KUKA KRL program: f1_Kuka_APT210T02S10.SRC

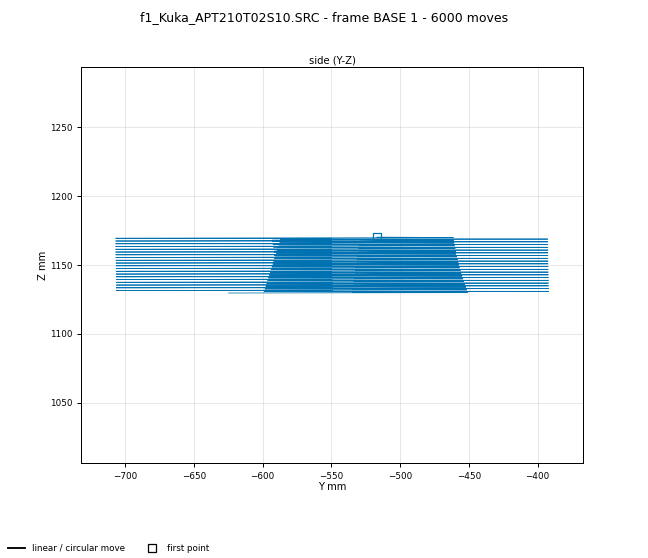
[picture p0: tool path of f1_Kuka_APT210T02S10.SRC in frame BASE 1, 6000 of 6001 moves have a stored position in this frame; points joined in program order, loops and branches not executed]
&ACCESS RVP
&REL 2
&PARAM TEMPLATE = C:\KRC\Roboter\Template\vorgabe
&PARAM EDITMASK = *
DEF f1_Kuka_APT210T02S10()


;FOLD INI;%{PE}%V3.2.0,%MKUKATPBASIS,%CINIT,%VCOMMON,%P
  ;FOLD BAS INI;%{E}%V3.2.0,%MKUKATPBASIS,%CINIT,%VINIT,%P
    GLOBAL INTERRUPT DECL 3 WHEN $STOPMESS==TRUE DO IR_STOPM ( )
    INTERRUPT ON 3
    BAS (#INITMOV,0 )
  ;ENDFOLD (BAS INI)
  ;FOLD USER INI;%{E}%V3.2.0,%MKUKATPUSER,%CINIT,%VINIT,%P
    ;Make your modifications here
  ;ENDFOLD (USER INI)
;ENDFOLD (INI)


;*** Make Null PTP Move
  PTP $pos_act

;*** Auto Load The Correct TOOL Data
  $tool=tool_data[2]

;*** Auto Load The Correct BASE Data
  $base=base_data[1]

  $ADVANCE = 5

;*** Restate Last Velocity
MMPM(30000.0)
SetRPM(8000)
LIN {X -0.168,Y -516.836,Z 1170.287,A 0.000,B 0.000,C 90.000,E1 267.593} C_DIS
LIN {X 0.032,Y -515.961,Z 1170.278,A 0.000,B 0.000,C 90.000,E1 266.102} C_DIS
LIN {X -0.268,Y -514.882,Z 1170.270,A 0.000,B 0.000,C 90.000,E1 264.666} C_DIS
LIN {X -0.155,Y -513.023,Z 1170.259,A 0.000,B 0.000,C 90.000,E1 262.591} C_DIS
LIN {X 0.153,Y -511.888,Z 1170.252,A 0.000,B 0.000,C 90.000,E1 261.376} C_DIS
LIN {X -0.212,Y -509.655,Z 1170.239,A 0.000,B 0.000,C 90.000,E1 259.050} C_DIS
LIN {X 0.192,Y -508.384,Z 1170.231,A 0.000,B 0.000,C 90.000,E1 257.521} C_DIS
LIN {X -0.015,Y -506.651,Z 1170.219,A 0.000,B 0.000,C 90.000,E1 255.463} C_DIS
LIN {X -0.094,Y -505.142,Z 1170.209,A 0.000,B 0.000,C 90.000,E1 253.685} C_DIS
LIN {X 0.005,Y -503.268,Z 1170.198,A 0.000,B 0.000,C 90.000,E1 251.583} C_DIS
LIN {X 0.305,Y -501.633,Z 1170.188,A 0.000,B 0.000,C 90.000,E1 249.752} C_DIS
LIN {X 0.102,Y -499.916,Z 1170.178,A 0.000,B 0.000,C 90.000,E1 247.975} C_DIS
LIN {X -0.084,Y -498.784,Z 1170.171,A 0.000,B 0.000,C 90.000,E1 246.794} C_DIS
LIN {X 0.030,Y -496.635,Z 1170.161,A 0.000,B 0.000,C 90.000,E1 244.973} C_DIS
LIN {X -0.003,Y -495.127,Z 1170.154,A 0.000,B 0.000,C 90.000,E1 243.768} C_DIS
LIN {X -0.213,Y -492.694,Z 1170.144,A 0.000,B 0.000,C 90.000,E1 241.975} C_DIS
LIN {X 0.240,Y -489.792,Z 1170.132,A 0.000,B 0.000,C 90.000,E1 239.793} C_DIS
LIN {X -0.045,Y -487.193,Z 1170.122,A 0.000,B 0.000,C 90.000,E1 237.995} C_DIS
LIN {X 0.307,Y -484.902,Z 1170.114,A 0.000,B 0.000,C 90.000,E1 236.421} C_DIS
LIN {X -0.151,Y -481.804,Z 1170.102,A 0.000,B 0.000,C 90.000,E1 234.322} C_DIS
LIN {X 0.167,Y -480.053,Z 1170.095,A 0.000,B 0.000,C 90.000,E1 233.050} C_DIS
LIN {X -0.126,Y -477.814,Z 1170.086,A 0.000,B 0.000,C 90.000,E1 231.537} C_DIS
LIN {X -0.166,Y -475.649,Z 1170.078,A 0.000,B 0.000,C 90.000,E1 229.989} C_DIS
LIN {X 0.056,Y -473.594,Z 1170.069,A 0.000,B 0.000,C 90.000,E1 228.405} C_DIS
LIN {X -0.073,Y -472.656,Z 1170.066,A 0.000,B 0.000,C 90.000,E1 227.796} C_DIS
LIN {X 0.019,Y -466.553,Z 1170.043,A 0.000,B 0.000,C 90.000,E1 223.704} C_DIS
LIN {X -0.010,Y -463.777,Z 1170.027,A 0.000,B 0.000,C 90.000,E1 220.862} C_DIS
LIN {X 0.041,Y -462.198,Z 1170.009,A 0.000,B 0.000,C 90.000,E1 217.684} C_DIS
LIN {X -0.051,Y -461.506,Z 1169.997,A 0.000,B 0.000,C 90.000,E1 215.471} C_DIS
LIN {X -0.057,Y -461.302,Z 1169.979,A 0.000,B 0.000,C 90.000,E1 212.291} C_DIS
LIN {X -0.265,Y -463.211,Z 1169.960,A 0.000,B 0.000,C 90.000,E1 208.821} C_DIS
LIN {X 0.242,Y -467.166,Z 1169.937,A 0.000,B 0.000,C 90.000,E1 204.643} C_DIS
LIN {X -0.175,Y -473.967,Z 1169.914,A 0.000,B 0.000,C 90.000,E1 200.610} C_DIS
LIN {X 0.182,Y -481.265,Z 1169.897,A 0.000,B 0.000,C 90.000,E1 197.457} C_DIS
LIN {X 0.057,Y -488.321,Z 1169.883,A 0.000,B 0.000,C 90.000,E1 195.009} C_DIS
LIN {X 0.091,Y -494.167,Z 1169.873,A 0.000,B 0.000,C 90.000,E1 193.175} C_DIS
LIN {X 0.040,Y -500.228,Z 1169.863,A 0.000,B 0.000,C 90.000,E1 191.366} C_DIS
LIN {X 0.024,Y -508.467,Z 1169.850,A 0.000,B 0.000,C 90.000,E1 188.973} C_DIS
LIN {X 0.172,Y -513.875,Z 1169.842,A 0.000,B 0.000,C 90.000,E1 187.473} C_DIS
LIN {X -0.083,Y -519.141,Z 1169.833,A 0.000,B 0.000,C 90.000,E1 186.030} C_DIS
LIN {X 0.214,Y -526.425,Z 1169.822,A 0.000,B 0.000,C 90.000,E1 183.955} C_DIS
LIN {X 0.093,Y -531.627,Z 1169.814,A 0.000,B 0.000,C 90.000,E1 182.522} C_DIS
LIN {X 0.067,Y -536.700,Z 1169.806,A 0.000,B 0.000,C 90.000,E1 181.088} C_DIS
LIN {X 0.146,Y -542.917,Z 1169.797,A 0.000,B 0.000,C 90.000,E1 179.370} C_DIS
LIN {X -0.219,Y -548.050,Z 1169.789,A 0.000,B 0.000,C 90.000,E1 177.993} C_DIS
LIN {X 0.003,Y -552.105,Z 1169.782,A 0.000,B 0.000,C 90.000,E1 176.846} C_DIS
LIN {X -0.088,Y -558.170,Z 1169.773,A 0.000,B 0.000,C 90.000,E1 175.179} C_DIS
LIN {X -0.149,Y -563.203,Z 1169.766,A 0.000,B 0.000,C 90.000,E1 173.799} C_DIS
LIN {X 0.032,Y -569.210,Z 1169.756,A 0.000,B 0.000,C 90.000,E1 172.129} C_DIS
LIN {X -0.066,Y -575.096,Z 1169.747,A 0.000,B 0.000,C 90.000,E1 170.500} C_DIS
LIN {X 0.100,Y -579.011,Z 1169.741,A 0.000,B 0.000,C 90.000,E1 169.398} C_DIS
LIN {X 0.330,Y -584.760,Z 1169.732,A 0.000,B 0.000,C 90.000,E1 167.757} C_DIS
LIN {X 0.109,Y -590.326,Z 1169.723,A 0.000,B 0.000,C 90.000,E1 166.172} C_DIS
LIN {X -0.136,Y -594.851,Z 1169.716,A 0.000,B 0.000,C 90.000,E1 164.866} C_DIS
LIN {X -0.020,Y -600.177,Z 1169.707,A 0.000,B 0.000,C 90.000,E1 163.268} C_DIS
LIN {X -0.023,Y -605.216,Z 1169.698,A 0.000,B 0.000,C 90.000,E1 161.692} C_DIS
LIN {X 0.153,Y -609.204,Z 1169.691,A 0.000,B 0.000,C 90.000,E1 160.369} C_DIS
LIN {X 0.024,Y -613.096,Z 1169.684,A 0.000,B 0.000,C 90.000,E1 159.082} C_DIS
LIN {X -0.011,Y -616.070,Z 1169.678,A 0.000,B 0.000,C 90.000,E1 158.050} C_DIS
LIN {X 0.178,Y -621.128,Z 1169.668,A 0.000,B 0.000,C 90.000,E1 156.230} C_DIS
LIN {X -0.085,Y -624.638,Z 1169.661,A 0.000,B 0.000,C 90.000,E1 154.973} C_DIS
LIN {X -0.002,Y -628.684,Z 1169.652,A 0.000,B 0.000,C 90.000,E1 153.435} C_DIS
LIN {X 0.131,Y -631.934,Z 1169.645,A 0.000,B 0.000,C 90.000,E1 152.153} C_DIS
LIN {X -0.248,Y -635.074,Z 1169.638,A 0.000,B 0.000,C 90.000,E1 150.923} C_DIS
LIN {X -0.271,Y -638.014,Z 1169.631,A 0.000,B 0.000,C 90.000,E1 149.665} C_DIS
LIN {X -0.247,Y -640.798,Z 1169.624,A 0.000,B 0.000,C 90.000,E1 148.408} C_DIS
LIN {X 0.154,Y -643.357,Z 1169.617,A 0.000,B 0.000,C 90.000,E1 147.120} C_DIS
LIN {X 0.059,Y -645.689,Z 1169.610,A 0.000,B 0.000,C 90.000,E1 145.881} C_DIS
LIN {X -0.102,Y -648.344,Z 1169.602,A 0.000,B 0.000,C 90.000,E1 144.402} C_DIS
LIN {X -0.180,Y -650.116,Z 1169.597,A 0.000,B 0.000,C 90.000,E1 143.417} C_DIS
LIN {X -0.314,Y -652.223,Z 1169.590,A 0.000,B 0.000,C 90.000,E1 142.190} C_DIS
LIN {X -0.069,Y -655.747,Z 1169.579,A 0.000,B 0.000,C 90.000,E1 140.194} C_DIS
LIN {X 0.299,Y -658.194,Z 1169.572,A 0.000,B 0.000,C 90.000,E1 138.933} C_DIS
LIN {X 0.206,Y -660.787,Z 1169.565,A 0.000,B 0.000,C 90.000,E1 137.715} C_DIS
LIN {X -0.364,Y -664.336,Z 1169.556,A 0.000,B 0.000,C 90.000,E1 136.053} C_DIS
LIN {X -0.380,Y -669.027,Z 1169.544,A 0.000,B 0.000,C 90.000,E1 133.866} C_DIS
LIN {X -0.255,Y -673.610,Z 1169.533,A 0.000,B 0.000,C 90.000,E1 131.919} C_DIS
LIN {X -0.295,Y -680.008,Z 1169.518,A 0.000,B 0.000,C 90.000,E1 129.277} C_DIS
LIN {X 0.098,Y -683.547,Z 1169.510,A 0.000,B 0.000,C 90.000,E1 127.810} C_DIS
LIN {X -0.031,Y -686.544,Z 1169.504,A 0.000,B 0.000,C 90.000,E1 126.629} C_DIS
LIN {X 0.221,Y -690.089,Z 1169.496,A 0.000,B 0.000,C 90.000,E1 125.185} C_DIS
LIN {X 0.129,Y -692.356,Z 1169.490,A 0.000,B 0.000,C 90.000,E1 124.246} C_DIS
LIN {X -0.110,Y -695.074,Z 1169.484,A 0.000,B 0.000,C 90.000,E1 123.086} C_DIS
LIN {X 0.287,Y -697.651,Z 1169.477,A 0.000,B 0.000,C 90.000,E1 121.878} C_DIS
LIN {X 0.130,Y -699.920,Z 1169.471,A 0.000,B 0.000,C 90.000,E1 120.718} C_DIS
LIN {X -0.021,Y -701.642,Z 1169.466,A 0.000,B 0.000,C 90.000,E1 119.795} C_DIS
LIN {X -0.211,Y -704.040,Z 1169.458,A 0.000,B 0.000,C 90.000,E1 118.409} C_DIS
LIN {X -0.022,Y -705.472,Z 1169.453,A 0.000,B 0.000,C 90.000,E1 117.462} C_DIS
LIN {X 0.224,Y -706.154,Z 1169.449,A 0.000,B 0.000,C 90.000,E1 116.744} C_DIS
LIN {X -0.182,Y -706.639,Z 1169.444,A 0.000,B 0.000,C 90.000,E1 115.848} C_DIS
LIN {X -0.241,Y -706.750,Z 1169.440,A 0.000,B 0.000,C 90.000,E1 115.155} C_DIS
LIN {X 0.348,Y -706.508,Z 1169.437,A 0.000,B 0.000,C 90.000,E1 114.643} C_DIS
LIN {X -0.296,Y -706.272,Z 1169.436,A 0.000,B 0.000,C 90.000,E1 114.463} C_DIS
LIN {X 0.287,Y -705.354,Z 1169.433,A 0.000,B 0.000,C 90.000,E1 113.951} C_DIS
LIN {X -0.354,Y -704.477,Z 1169.432,A 0.000,B 0.000,C 90.000,E1 113.770} C_DIS
LIN {X 0.213,Y -702.290,Z 1169.429,A 0.000,B 0.000,C 90.000,E1 113.259} C_DIS
LIN {X 0.075,Y -701.376,Z 1169.429,A 0.000,B 0.000,C 90.000,E1 113.153} C_DIS
LIN {X -0.030,Y -696.702,Z 1169.426,A 0.000,B 0.000,C 90.000,E1 112.695} C_DIS
LIN {X -0.167,Y -694.978,Z 1169.425,A 0.000,B 0.000,C 90.000,E1 112.589} C_DIS
LIN {X 0.211,Y -692.477,Z 1169.425,A 0.000,B 0.000,C 90.000,E1 112.461} C_DIS
LIN {X -0.061,Y -685.884,Z 1169.424,A 0.000,B 0.000,C 90.000,E1 112.280} C_DIS
LIN {X -0.050,Y -684.884,Z 1169.424,A 0.000,B 0.000,C 90.000,E1 112.259} C_DIS
LIN {X 0.023,Y -677.229,Z 1169.423,A 0.000,B 0.000,C 90.000,E1 112.206} C_DIS
LIN {X -0.028,Y -604.897,Z 1169.423,A 0.000,B 0.000,C 90.000,E1 112.206} C_DIS
LIN {X -0.262,Y -599.969,Z 1169.422,A 0.000,B 0.000,C 90.000,E1 111.897} C_DIS
LIN {X 0.216,Y -595.825,Z 1169.420,A 0.000,B 0.000,C 90.000,E1 111.535} C_DIS
LIN {X 0.002,Y -584.117,Z 1169.414,A 0.000,B 0.000,C 90.000,E1 110.556} C_DIS
LIN {X -0.067,Y -577.421,Z 1169.411,A 0.000,B 0.000,C 90.000,E1 109.993} C_DIS
LIN {X -0.058,Y -574.631,Z 1169.410,A 0.000,B 0.000,C 90.000,E1 109.758} C_DIS
LIN {X -0.102,Y -568.886,Z 1169.407,A 0.000,B 0.000,C 90.000,E1 109.322} C_DIS
LIN {X -0.058,Y -561.036,Z 1169.404,A 0.000,B 0.000,C 90.000,E1 108.779} C_DIS
LIN {X -0.036,Y -556.428,Z 1169.403,A 0.000,B 0.000,C 90.000,E1 108.471} C_DIS
LIN {X 0.260,Y -551.811,Z 1169.401,A 0.000,B 0.000,C 90.000,E1 108.055} C_DIS
LIN {X -0.164,Y -550.478,Z 1169.399,A 0.000,B 0.000,C 90.000,E1 107.873} C_DIS
LIN {X -0.206,Y -550.464,Z 1169.399,A 0.000,B 0.000,C 90.000,E1 107.873} C_DIS
LIN {X 0.054,Y -550.010,Z 1169.397,A 0.000,B 0.000,C 90.000,E1 107.457} C_DIS
LIN {X 0.084,Y -550.645,Z 1169.391,A 0.000,B 0.000,C 90.000,E1 106.441} C_DIS
LIN {X 0.127,Y -551.600,Z 1169.385,A 0.000,B 0.000,C 90.000,E1 105.315} C_DIS
LIN {X 0.139,Y -553.320,Z 1169.374,A 0.000,B 0.000,C 90.000,E1 103.355} C_DIS
LIN {X -0.070,Y -555.144,Z 1169.364,A 0.000,B 0.000,C 90.000,E1 101.422} C_DIS
LIN {X 0.213,Y -557.116,Z 1169.353,A 0.000,B 0.000,C 90.000,E1 99.443} C_DIS
LIN {X -0.156,Y -558.706,Z 1169.343,A 0.000,B 0.000,C 90.000,E1 97.814} C_DIS
LIN {X 0.252,Y -559.602,Z 1169.337,A 0.000,B 0.000,C 90.000,E1 96.663} C_DIS
LIN {X -0.219,Y -560.844,Z 1169.328,A 0.000,B 0.000,C 90.000,E1 95.049} C_DIS
LIN {X 0.164,Y -562.571,Z 1169.314,A 0.000,B 0.000,C 90.000,E1 92.522} C_DIS
LIN {X -0.224,Y -564.025,Z 1169.303,A 0.000,B 0.000,C 90.000,E1 90.630} C_DIS
LIN {X 0.211,Y -564.856,Z 1169.297,A 0.000,B 0.000,C 90.000,E1 89.484} C_DIS
LIN {X 0.216,Y -565.746,Z 1169.290,A 0.000,B 0.000,C 90.000,E1 88.108} C_DIS
LIN {X -0.208,Y -566.791,Z 1169.281,A 0.000,B 0.000,C 90.000,E1 86.502} C_DIS
LIN {X 0.142,Y -568.012,Z 1169.270,A 0.000,B 0.000,C 90.000,E1 84.546} C_DIS
LIN {X -0.151,Y -569.120,Z 1169.261,A 0.000,B 0.000,C 90.000,E1 82.932} C_DIS
LIN {X 0.309,Y -569.631,Z 1169.256,A 0.000,B 0.000,C 90.000,E1 82.064} C_DIS
LIN {X -0.072,Y -570.396,Z 1169.249,A 0.000,B 0.000,C 90.000,E1 80.735} C_DIS
LIN {X 0.206,Y -571.081,Z 1169.241,A 0.000,B 0.000,C 90.000,E1 79.342} C_DIS
LIN {X 0.044,Y -571.783,Z 1169.233,A 0.000,B 0.000,C 90.000,E1 77.993} C_DIS
LIN {X -0.105,Y -572.436,Z 1169.226,A 0.000,B 0.000,C 90.000,E1 76.645} C_DIS
LIN {X -0.108,Y -573.167,Z 1169.218,A 0.000,B 0.000,C 90.000,E1 75.283} C_DIS
LIN {X -0.114,Y -574.441,Z 1169.205,A 0.000,B 0.000,C 90.000,E1 72.834} C_DIS
LIN {X -0.286,Y -575.459,Z 1169.196,A 0.000,B 0.000,C 90.000,E1 71.221} C_DIS
LIN {X -0.072,Y -576.669,Z 1169.187,A 0.000,B 0.000,C 90.000,E1 69.571} C_DIS
LIN {X 0.248,Y -578.771,Z 1169.173,A 0.000,B 0.000,C 90.000,E1 67.102} C_DIS
LIN {X -0.033,Y -579.878,Z 1169.167,A 0.000,B 0.000,C 90.000,E1 66.049} C_DIS
LIN {X 0.188,Y -581.373,Z 1169.158,A 0.000,B 0.000,C 90.000,E1 64.409} C_DIS
LIN {X 0.048,Y -583.149,Z 1169.147,A 0.000,B 0.000,C 90.000,E1 62.538} C_DIS
LIN {X 0.074,Y -584.629,Z 1169.139,A 0.000,B 0.000,C 90.000,E1 60.923} C_DIS
LIN {X -0.101,Y -586.035,Z 1169.130,A 0.000,B 0.000,C 90.000,E1 59.331} C_DIS
LIN {X -0.125,Y -587.060,Z 1169.122,A 0.000,B 0.000,C 90.000,E1 57.995} C_DIS
LIN {X 0.049,Y -588.178,Z 1169.113,A 0.000,B 0.000,C 90.000,E1 56.373} C_DIS
LIN {X -0.184,Y -588.691,Z 1169.109,A 0.000,B 0.000,C 90.000,E1 55.595} C_DIS
LIN {X 0.278,Y -589.415,Z 1169.103,A 0.000,B 0.000,C 90.000,E1 54.482} C_DIS
LIN {X 0.060,Y -590.570,Z 1169.093,A 0.000,B 0.000,C 90.000,E1 52.637} C_DIS
LIN {X -0.032,Y -591.823,Z 1169.081,A 0.000,B 0.000,C 90.000,E1 50.517} C_DIS
LIN {X -0.106,Y -592.247,Z 1169.075,A 0.000,B 0.000,C 90.000,E1 49.461} C_DIS
LIN {X 0.029,Y -592.618,Z 1169.067,A 0.000,B 0.000,C 90.000,E1 48.119} C_DIS
LIN {X 0.122,Y -592.831,Z 1169.060,A 0.000,B 0.000,C 90.000,E1 46.782} C_DIS
LIN {X 0.027,Y -592.788,Z 1169.054,A 0.000,B 0.000,C 90.000,E1 45.729} C_DIS
LIN {X -0.295,Y -592.486,Z 1169.047,A 0.000,B 0.000,C 90.000,E1 44.433} C_DIS
LIN {X -0.159,Y -592.177,Z 1169.042,A 0.000,B 0.000,C 90.000,E1 43.623} C_DIS
LIN {X 0.166,Y -591.591,Z 1169.036,A 0.000,B 0.000,C 90.000,E1 42.528} C_DIS
LIN {X 0.088,Y -590.864,Z 1169.031,A 0.000,B 0.000,C 90.000,E1 41.472} C_DIS
LIN {X 0.005,Y -589.930,Z 1169.025,A 0.000,B 0.000,C 90.000,E1 40.415} C_DIS
LIN {X 0.110,Y -588.475,Z 1169.017,A 0.000,B 0.000,C 90.000,E1 39.072} C_DIS
LIN {X -0.213,Y -587.458,Z 1169.013,A 0.000,B 0.000,C 90.000,E1 38.302} C_DIS
LIN {X -0.256,Y -585.940,Z 1169.007,A 0.000,B 0.000,C 90.000,E1 37.237} C_DIS
LIN {X 0.032,Y -584.075,Z 1169.001,A 0.000,B 0.000,C 90.000,E1 36.137} C_DIS
LIN {X 0.056,Y -582.983,Z 1168.998,A 0.000,B 0.000,C 90.000,E1 35.598} C_DIS
LIN {X -0.050,Y -580.579,Z 1168.992,A 0.000,B 0.000,C 90.000,E1 34.532} C_DIS
LIN {X -0.040,Y -579.112,Z 1168.989,A 0.000,B 0.000,C 90.000,E1 33.992} C_DIS
LIN {X 0.107,Y -574.932,Z 1168.981,A 0.000,B 0.000,C 90.000,E1 32.625} C_DIS
LIN {X 0.084,Y -572.991,Z 1168.978,A 0.000,B 0.000,C 90.000,E1 32.084} C_DIS
LIN {X 0.171,Y -569.582,Z 1168.974,A 0.000,B 0.000,C 90.000,E1 31.258} C_DIS
LIN {X -0.167,Y -565.336,Z 1168.969,A 0.000,B 0.000,C 90.000,E1 30.335} C_DIS
LIN {X 0.032,Y -561.090,Z 1168.964,A 0.000,B 0.000,C 90.000,E1 29.489} C_DIS
LIN {X -0.096,Y -558.078,Z 1168.961,A 0.000,B 0.000,C 90.000,E1 28.949} C_DIS
LIN {X -0.086,Y -552.377,Z 1168.955,A 0.000,B 0.000,C 90.000,E1 27.975} C_DIS
LIN {X 0.086,Y -547.919,Z 1168.952,A 0.000,B 0.000,C 90.000,E1 27.257} C_DIS
LIN {X 0.094,Y -544.067,Z 1168.948,A 0.000,B 0.000,C 90.000,E1 26.693} C_DIS
LIN {X -0.169,Y -539.974,Z 1168.945,A 0.000,B 0.000,C 90.000,E1 26.155} C_DIS
LIN {X -0.214,Y -535.555,Z 1168.942,A 0.000,B 0.000,C 90.000,E1 25.591} C_DIS
LIN {X 0.051,Y -529.716,Z 1168.938,A 0.000,B 0.000,C 90.000,E1 24.847} C_DIS
LIN {X 0.113,Y -523.679,Z 1168.934,A 0.000,B 0.000,C 90.000,E1 24.131} C_DIS
LIN {X 0.093,Y -514.571,Z 1168.929,A 0.000,B 0.000,C 90.000,E1 23.131} C_DIS
LIN {X -0.134,Y -509.137,Z 1168.925,A 0.000,B 0.000,C 90.000,E1 22.589} C_DIS
LIN {X 0.231,Y -500.761,Z 1168.921,A 0.000,B 0.000,C 90.000,E1 21.716} C_DIS
LIN {X 0.086,Y -490.782,Z 1168.916,A 0.000,B 0.000,C 90.000,E1 20.791} C_DIS
LIN {X -0.095,Y -480.589,Z 1168.910,A 0.000,B 0.000,C 90.000,E1 19.885} C_DIS
LIN {X 0.010,Y -470.428,Z 1168.905,A 0.000,B 0.000,C 90.000,E1 18.960} C_DIS
LIN {X -0.086,Y -458.727,Z 1168.900,A 0.000,B 0.000,C 90.000,E1 17.928} C_DIS
LIN {X 0.121,Y -447.291,Z 1168.894,A 0.000,B 0.000,C 90.000,E1 16.858} C_DIS
LIN {X -0.016,Y -428.509,Z 1168.883,A 0.000,B 0.000,C 90.000,E1 15.009} C_DIS
LIN {X -0.007,Y -416.177,Z 1168.876,A 0.000,B 0.000,C 90.000,E1 13.647} C_DIS
LIN {X 0.070,Y -407.100,Z 1168.870,A 0.000,B 0.000,C 90.000,E1 12.535} C_DIS
LIN {X 0.182,Y -399.418,Z 1168.864,A 0.000,B 0.000,C 90.000,E1 11.478} C_DIS
LIN {X 0.126,Y -396.306,Z 1168.861,A 0.000,B 0.000,C 90.000,E1 11.007} C_DIS
LIN {X -0.144,Y -393.394,Z 1168.858,A 0.000,B 0.000,C 90.000,E1 10.423} C_DIS
LIN {X 0.166,Y -392.697,Z 1168.856,A 0.000,B 0.000,C 90.000,E1 10.018} C_DIS
LIN {X 0.128,Y -392.689,Z 1168.856,A 0.000,B 0.000,C 90.000,E1 10.018} C_DIS
LIN {X -0.059,Y -393.219,Z 1168.853,A 0.000,B 0.000,C 90.000,E1 9.613} C_DIS
LIN {X -0.141,Y -394.979,Z 1168.849,A 0.000,B 0.000,C 90.000,E1 8.916} C_DIS
LIN {X 0.138,Y -397.945,Z 1168.845,A 0.000,B 0.000,C 90.000,E1 7.992} C_DIS
LIN {X -0.024,Y -402.282,Z 1168.839,A 0.000,B 0.000,C 90.000,E1 7.004} C_DIS
LIN {X -0.019,Y -407.163,Z 1168.835,A 0.000,B 0.000,C 90.000,E1 6.258} C_DIS
LIN {X 0.161,Y -410.505,Z 1168.833,A 0.000,B 0.000,C 90.000,E1 5.910} C_DIS
LIN {X 0.103,Y -415.574,Z 1168.831,A 0.000,B 0.000,C 90.000,E1 5.511} C_DIS
LIN {X -0.051,Y -426.674,Z 1168.826,A 0.000,B 0.000,C 90.000,E1 4.702} C_DIS
LIN {X 0.136,Y -449.122,Z 1168.817,A 0.000,B 0.000,C 90.000,E1 3.037} C_DIS
LIN {X -0.172,Y -465.211,Z 1168.811,A 0.000,B 0.000,C 90.000,E1 1.949} C_DIS
LIN {X -0.008,Y -474.614,Z 1168.807,A 0.000,B 0.000,C 90.000,E1 1.260} C_DIS
LIN {X 0.001,Y -482.394,Z 1168.804,A 0.000,B 0.000,C 90.000,E1 0.688} C_DIS
LIN {X 0.000,Y -491.215,Z 1168.800,A 0.000,B 0.000,C 90.000,E1 360.000} C_DIS
LIN {X 0.020,Y -496.714,Z 1168.797,A 0.000,B 0.000,C 90.000,E1 359.542} C_DIS
LIN {X -0.079,Y -503.698,Z 1168.794,A 0.000,B 0.000,C 90.000,E1 358.912} C_DIS
LIN {X -0.030,Y -510.446,Z 1168.790,A 0.000,B 0.000,C 90.000,E1 358.224} C_DIS
LIN {X -0.184,Y -516.881,Z 1168.786,A 0.000,B 0.000,C 90.000,E1 357.535} C_DIS
LIN {X -0.024,Y -523.035,Z 1168.782,A 0.000,B 0.000,C 90.000,E1 356.788} C_DIS
LIN {X -0.268,Y -528.498,Z 1168.778,A 0.000,B 0.000,C 90.000,E1 356.102} C_DIS
LIN {X -0.038,Y -533.541,Z 1168.774,A 0.000,B 0.000,C 90.000,E1 355.355} C_DIS
LIN {X -0.021,Y -537.235,Z 1168.771,A 0.000,B 0.000,C 90.000,E1 354.780} C_DIS
LIN {X 0.024,Y -540.612,Z 1168.768,A 0.000,B 0.000,C 90.000,E1 354.204} C_DIS
LIN {X -0.170,Y -544.359,Z 1168.764,A 0.000,B 0.000,C 90.000,E1 353.514} C_DIS
LIN {X 0.273,Y -547.796,Z 1168.760,A 0.000,B 0.000,C 90.000,E1 352.761} C_DIS
LIN {X -0.151,Y -550.453,Z 1168.757,A 0.000,B 0.000,C 90.000,E1 352.243} C_DIS
LIN {X 0.096,Y -553.870,Z 1168.752,A 0.000,B 0.000,C 90.000,E1 351.376} C_DIS
LIN {X -0.211,Y -555.963,Z 1168.749,A 0.000,B 0.000,C 90.000,E1 350.849} C_DIS
LIN {X 0.233,Y -559.687,Z 1168.743,A 0.000,B 0.000,C 90.000,E1 349.690} C_DIS
LIN {X 0.279,Y -562.974,Z 1168.737,A 0.000,B 0.000,C 90.000,E1 348.578} C_DIS
LIN {X -0.176,Y -565.979,Z 1168.731,A 0.000,B 0.000,C 90.000,E1 347.521} C_DIS
LIN {X 0.137,Y -569.476,Z 1168.723,A 0.000,B 0.000,C 90.000,E1 346.117} C_DIS
LIN {X 0.088,Y -572.689,Z 1168.715,A 0.000,B 0.000,C 90.000,E1 344.755} C_DIS
LIN {X 0.257,Y -574.483,Z 1168.711,A 0.000,B 0.000,C 90.000,E1 343.921} C_DIS
LIN {X -0.097,Y -577.404,Z 1168.703,A 0.000,B 0.000,C 90.000,E1 342.598} C_DIS
LIN {X 0.119,Y -579.072,Z 1168.699,A 0.000,B 0.000,C 90.000,E1 341.764} C_DIS
LIN {X 0.027,Y -581.631,Z 1168.691,A 0.000,B 0.000,C 90.000,E1 340.423} C_DIS
LIN {X 0.125,Y -583.415,Z 1168.685,A 0.000,B 0.000,C 90.000,E1 339.337} C_DIS
LIN {X -0.095,Y -584.891,Z 1168.679,A 0.000,B 0.000,C 90.000,E1 338.284} C_DIS
LIN {X -0.165,Y -585.825,Z 1168.675,A 0.000,B 0.000,C 90.000,E1 337.486} C_DIS
LIN {X 0.124,Y -586.340,Z 1168.672,A 0.000,B 0.000,C 90.000,E1 336.922} C_DIS
LIN {X 0.299,Y -586.806,Z 1168.667,A 0.000,B 0.000,C 90.000,E1 336.102} C_DIS
LIN {X -0.179,Y -587.004,Z 1168.664,A 0.000,B 0.000,C 90.000,E1 335.613} C_DIS
LIN {X -0.114,Y -586.849,Z 1168.659,A 0.000,B 0.000,C 90.000,E1 334.537} C_DIS
LIN {X 0.063,Y -586.397,Z 1168.654,A 0.000,B 0.000,C 90.000,E1 333.717} C_DIS
LIN {X 0.092,Y -585.896,Z 1168.651,A 0.000,B 0.000,C 90.000,E1 333.179} C_DIS
LIN {X 0.256,Y -584.870,Z 1168.647,A 0.000,B 0.000,C 90.000,E1 332.359} C_DIS
LIN {X 0.036,Y -582.987,Z 1168.641,A 0.000,B 0.000,C 90.000,E1 331.307} C_DIS
LIN {X -0.206,Y -580.282,Z 1168.635,A 0.000,B 0.000,C 90.000,E1 330.255} C_DIS
LIN {X 0.160,Y -577.838,Z 1168.630,A 0.000,B 0.000,C 90.000,E1 329.410} C_DIS
LIN {X -0.004,Y -574.491,Z 1168.626,A 0.000,B 0.000,C 90.000,E1 328.614} C_DIS
LIN {X 0.181,Y -571.023,Z 1168.622,A 0.000,B 0.000,C 90.000,E1 327.916} C_DIS
LIN {X -0.072,Y -565.352,Z 1168.617,A 0.000,B 0.000,C 90.000,E1 326.993} C_DIS
LIN {X -0.067,Y -562.612,Z 1168.614,A 0.000,B 0.000,C 90.000,E1 326.580} C_DIS
LIN {X 0.129,Y -558.615,Z 1168.611,A 0.000,B 0.000,C 90.000,E1 326.008} C_DIS
LIN {X -0.016,Y -554.424,Z 1168.608,A 0.000,B 0.000,C 90.000,E1 325.468} C_DIS
LIN {X -0.065,Y -551.036,Z 1168.606,A 0.000,B 0.000,C 90.000,E1 325.055} C_DIS
LIN {X 0.097,Y -543.692,Z 1168.601,A 0.000,B 0.000,C 90.000,E1 324.196} C_DIS
LIN {X -0.179,Y -531.199,Z 1168.594,A 0.000,B 0.000,C 90.000,E1 322.844} C_DIS
LIN {X 0.071,Y -525.417,Z 1168.590,A 0.000,B 0.000,C 90.000,E1 322.145} C_DIS
LIN {X 0.185,Y -522.185,Z 1168.587,A 0.000,B 0.000,C 90.000,E1 321.698} C_DIS
LIN {X 0.004,Y -519.752,Z 1168.585,A 0.000,B 0.000,C 90.000,E1 321.251} C_DIS
LIN {X 0.220,Y -517.837,Z 1168.582,A 0.000,B 0.000,C 90.000,E1 320.642} C_DIS
LIN {X -0.097,Y -516.894,Z 1168.577,A 0.000,B 0.000,C 90.000,E1 319.908} C_DIS
LIN {X 0.033,Y -516.898,Z 1168.572,A 0.000,B 0.000,C 90.000,E1 319.013} C_DIS
LIN {X -0.207,Y -517.985,Z 1168.561,A 0.000,B 0.000,C 90.000,E1 316.986} C_DIS
LIN {X 0.107,Y -518.780,Z 1168.553,A 0.000,B 0.000,C 90.000,E1 315.486} C_DIS
LIN {X -0.100,Y -519.889,Z 1168.541,A 0.000,B 0.000,C 90.000,E1 313.461} C_DIS
LIN {X 0.122,Y -521.066,Z 1168.530,A 0.000,B 0.000,C 90.000,E1 311.391} C_DIS
LIN {X 0.138,Y -521.966,Z 1168.522,A 0.000,B 0.000,C 90.000,E1 309.930} C_DIS
LIN {X 0.188,Y -523.013,Z 1168.512,A 0.000,B 0.000,C 90.000,E1 308.177} C_DIS
LIN {X -0.054,Y -524.076,Z 1168.503,A 0.000,B 0.000,C 90.000,E1 306.457} C_DIS
LIN {X 0.076,Y -525.342,Z 1168.490,A 0.000,B 0.000,C 90.000,E1 304.119} C_DIS
LIN {X -0.287,Y -526.458,Z 1168.480,A 0.000,B 0.000,C 90.000,E1 302.418} C_DIS
LIN {X -0.177,Y -527.438,Z 1168.470,A 0.000,B 0.000,C 90.000,E1 300.669} C_DIS
LIN {X -0.119,Y -527.893,Z 1168.465,A 0.000,B 0.000,C 90.000,E1 299.795} C_DIS
LIN {X 0.204,Y -528.484,Z 1168.456,A 0.000,B 0.000,C 90.000,E1 298.025} C_DIS
LIN {X -0.122,Y -528.799,Z 1168.448,A 0.000,B 0.000,C 90.000,E1 296.616} C_DIS
LIN {X -0.141,Y -528.955,Z 1168.441,A 0.000,B 0.000,C 90.000,E1 295.463} C_DIS
LIN {X 0.098,Y -529.006,Z 1168.435,A 0.000,B 0.000,C 90.000,E1 294.283} C_DIS
LIN {X -0.074,Y -528.949,Z 1168.424,A 0.000,B 0.000,C 90.000,E1 292.280} C_DIS
LIN {X -0.148,Y -528.670,Z 1168.414,A 0.000,B 0.000,C 90.000,E1 290.556} C_DIS
LIN {X 0.256,Y -528.273,Z 1168.405,A 0.000,B 0.000,C 90.000,E1 288.779} C_DIS
LIN {X 0.122,Y -527.880,Z 1168.398,A 0.000,B 0.000,C 90.000,E1 287.638} C_DIS
LIN {X -0.001,Y -527.371,Z 1168.390,A 0.000,B 0.000,C 90.000,E1 286.205} C_DIS
LIN {X -0.152,Y -526.839,Z 1168.384,A 0.000,B 0.000,C 90.000,E1 285.064} C_DIS
LIN {X 0.055,Y -526.156,Z 1168.377,A 0.000,B 0.000,C 90.000,E1 283.883} C_DIS
LIN {X 0.268,Y -525.334,Z 1168.369,A 0.000,B 0.000,C 90.000,E1 282.411} C_DIS
LIN {X -0.161,Y -524.370,Z 1168.361,A 0.000,B 0.000,C 90.000,E1 281.007} C_DIS
LIN {X -0.187,Y -523.397,Z 1168.353,A 0.000,B 0.000,C 90.000,E1 279.557} C_DIS
LIN {X -0.225,Y -522.458,Z 1168.345,A 0.000,B 0.000,C 90.000,E1 278.106} C_DIS
LIN {X 0.163,Y -521.408,Z 1168.335,A 0.000,B 0.000,C 90.000,E1 276.315} C_DIS
LIN {X -0.052,Y -520.424,Z 1168.326,A 0.000,B 0.000,C 90.000,E1 274.588} C_DIS
LIN {X 0.189,Y -519.608,Z 1168.316,A 0.000,B 0.000,C 90.000,E1 272.808} C_DIS
LIN {X -0.248,Y -518.576,Z 1168.303,A 0.000,B 0.000,C 90.000,E1 270.516} C_DIS
LIN {X -0.022,Y -517.919,Z 1168.295,A 0.000,B 0.000,C 90.000,E1 269.026} C_DIS
LIN {X -0.250,Y -517.425,Z 1168.288,A 0.000,B 0.000,C 90.000,E1 267.879} C_DIS
LIN {X -0.105,Y -516.392,Z 1168.278,A 0.000,B 0.000,C 90.000,E1 266.102} C_DIS
LIN {X 0.085,Y -515.122,Z 1168.269,A 0.000,B 0.000,C 90.000,E1 264.318} C_DIS
LIN {X 0.208,Y -513.182,Z 1168.257,A 0.000,B 0.000,C 90.000,E1 262.243} C_DIS
LIN {X 0.043,Y -512.324,Z 1168.252,A 0.000,B 0.000,C 90.000,E1 261.376} C_DIS
LIN {X 0.154,Y -509.809,Z 1168.237,A 0.000,B 0.000,C 90.000,E1 258.701} C_DIS
LIN {X 0.104,Y -508.764,Z 1168.231,A 0.000,B 0.000,C 90.000,E1 257.521} C_DIS
LIN {X -0.044,Y -507.309,Z 1168.221,A 0.000,B 0.000,C 90.000,E1 255.755} C_DIS
LIN {X -0.102,Y -505.787,Z 1168.211,A 0.000,B 0.000,C 90.000,E1 253.976} C_DIS
LIN {X -0.067,Y -504.713,Z 1168.204,A 0.000,B 0.000,C 90.000,E1 252.779} C_DIS
LIN {X 0.107,Y -503.060,Z 1168.194,A 0.000,B 0.000,C 90.000,E1 250.967} C_DIS
LIN {X 0.158,Y -501.679,Z 1168.186,A 0.000,B 0.000,C 90.000,E1 249.464} C_DIS
LIN {X 0.132,Y -500.018,Z 1168.176,A 0.000,B 0.000,C 90.000,E1 247.667} C_DIS
LIN {X -0.121,Y -499.139,Z 1168.171,A 0.000,B 0.000,C 90.000,E1 246.794} C_DIS
LIN {X 0.001,Y -496.962,Z 1168.161,A 0.000,B 0.000,C 90.000,E1 244.973} C_DIS
LIN {X 0.018,Y -495.018,Z 1168.153,A 0.000,B 0.000,C 90.000,E1 243.461} C_DIS
LIN {X 0.030,Y -492.590,Z 1168.143,A 0.000,B 0.000,C 90.000,E1 241.641} C_DIS
LIN {X 0.231,Y -490.079,Z 1168.132,A 0.000,B 0.000,C 90.000,E1 239.793} C_DIS
LIN {X 0.191,Y -487.011,Z 1168.120,A 0.000,B 0.000,C 90.000,E1 237.661} C_DIS
LIN {X 0.180,Y -483.775,Z 1168.109,A 0.000,B 0.000,C 90.000,E1 235.515} C_DIS
LIN {X -0.122,Y -481.157,Z 1168.098,A 0.000,B 0.000,C 90.000,E1 233.703} C_DIS
LIN {X 0.084,Y -478.441,Z 1168.088,A 0.000,B 0.000,C 90.000,E1 231.823} C_DIS
LIN {X 0.057,Y -476.206,Z 1168.079,A 0.000,B 0.000,C 90.000,E1 230.275} C_DIS
LIN {X 0.074,Y -473.704,Z 1168.069,A 0.000,B 0.000,C 90.000,E1 228.405} C_DIS
LIN {X 0.039,Y -472.211,Z 1168.064,A 0.000,B 0.000,C 90.000,E1 227.472} C_DIS
LIN {X 0.112,Y -466.186,Z 1168.041,A 0.000,B 0.000,C 90.000,E1 223.380} C_DIS
LIN {X -0.139,Y -463.119,Z 1168.022,A 0.000,B 0.000,C 90.000,E1 219.930} C_DIS
LIN {X 0.061,Y -462.042,Z 1168.009,A 0.000,B 0.000,C 90.000,E1 217.684} C_DIS
LIN {X -0.157,Y -461.368,Z 1167.999,A 0.000,B 0.000,C 90.000,E1 215.804} C_DIS
LIN {X 0.075,Y -461.025,Z 1167.978,A 0.000,B 0.000,C 90.000,E1 211.957} C_DIS
LIN {X -0.279,Y -462.693,Z 1167.960,A 0.000,B 0.000,C 90.000,E1 208.821} C_DIS
LIN {X 0.201,Y -466.585,Z 1167.937,A 0.000,B 0.000,C 90.000,E1 204.643} C_DIS
LIN {X -0.170,Y -472.217,Z 1167.918,A 0.000,B 0.000,C 90.000,E1 201.227} C_DIS
LIN {X 0.071,Y -476.133,Z 1167.907,A 0.000,B 0.000,C 90.000,E1 199.322} C_DIS
LIN {X -0.094,Y -483.327,Z 1167.892,A 0.000,B 0.000,C 90.000,E1 196.551} C_DIS
LIN {X -0.040,Y -492.787,Z 1167.875,A 0.000,B 0.000,C 90.000,E1 193.480} C_DIS
LIN {X -0.091,Y -499.858,Z 1167.863,A 0.000,B 0.000,C 90.000,E1 191.366} C_DIS
LIN {X -0.119,Y -508.171,Z 1167.850,A 0.000,B 0.000,C 90.000,E1 188.973} C_DIS
LIN {X 0.022,Y -513.582,Z 1167.842,A 0.000,B 0.000,C 90.000,E1 187.473} C_DIS
LIN {X -0.160,Y -517.857,Z 1167.835,A 0.000,B 0.000,C 90.000,E1 186.315} C_DIS
LIN {X 0.105,Y -524.111,Z 1167.825,A 0.000,B 0.000,C 90.000,E1 184.531} C_DIS
LIN {X -0.028,Y -529.358,Z 1167.817,A 0.000,B 0.000,C 90.000,E1 183.094} C_DIS
LIN {X -0.108,Y -533.505,Z 1167.811,A 0.000,B 0.000,C 90.000,E1 181.949} C_DIS
LIN {X -0.089,Y -539.726,Z 1167.801,A 0.000,B 0.000,C 90.000,E1 180.229} C_DIS
LIN {X 0.021,Y -544.884,Z 1167.793,A 0.000,B 0.000,C 90.000,E1 178.797} C_DIS
LIN {X 0.190,Y -549.066,Z 1167.787,A 0.000,B 0.000,C 90.000,E1 177.650} C_DIS
LIN {X 0.098,Y -556.173,Z 1167.776,A 0.000,B 0.000,C 90.000,E1 175.698} C_DIS
LIN {X 0.003,Y -561.287,Z 1167.768,A 0.000,B 0.000,C 90.000,E1 174.318} C_DIS
LIN {X 0.147,Y -567.335,Z 1167.759,A 0.000,B 0.000,C 90.000,E1 172.648} C_DIS
LIN {X -0.178,Y -572.356,Z 1167.752,A 0.000,B 0.000,C 90.000,E1 171.310} C_DIS
LIN {X -0.298,Y -578.297,Z 1167.743,A 0.000,B 0.000,C 90.000,E1 169.690} C_DIS
LIN {X -0.088,Y -584.159,Z 1167.734,A 0.000,B 0.000,C 90.000,E1 168.049} C_DIS
LIN {X 0.250,Y -589.739,Z 1167.725,A 0.000,B 0.000,C 90.000,E1 166.408} C_DIS
LIN {X -0.004,Y -594.341,Z 1167.717,A 0.000,B 0.000,C 90.000,E1 165.102} C_DIS
LIN {X 0.106,Y -599.716,Z 1167.708,A 0.000,B 0.000,C 90.000,E1 163.504} C_DIS
LIN {X -0.091,Y -604.769,Z 1167.700,A 0.000,B 0.000,C 90.000,E1 161.945} C_DIS
LIN {X 0.272,Y -608.812,Z 1167.692,A 0.000,B 0.000,C 90.000,E1 160.604} C_DIS
LIN {X -0.121,Y -613.460,Z 1167.684,A 0.000,B 0.000,C 90.000,E1 159.082} C_DIS
LIN {X 0.078,Y -616.393,Z 1167.678,A 0.000,B 0.000,C 90.000,E1 158.028} C_DIS
LIN {X 0.064,Y -619.942,Z 1167.671,A 0.000,B 0.000,C 90.000,E1 156.741} C_DIS
LIN {X -0.224,Y -623.510,Z 1167.664,A 0.000,B 0.000,C 90.000,E1 155.485} C_DIS
LIN {X -0.198,Y -626.258,Z 1167.658,A 0.000,B 0.000,C 90.000,E1 154.460} C_DIS
LIN {X -0.105,Y -629.575,Z 1167.651,A 0.000,B 0.000,C 90.000,E1 153.179} C_DIS
LIN {X 0.075,Y -633.388,Z 1167.643,A 0.000,B 0.000,C 90.000,E1 151.641} C_DIS
LIN {X -0.369,Y -635.222,Z 1167.638,A 0.000,B 0.000,C 90.000,E1 150.923} C_DIS
LIN {X 0.115,Y -637.578,Z 1167.633,A 0.000,B 0.000,C 90.000,E1 149.871} C_DIS
LIN {X 0.131,Y -640.355,Z 1167.626,A 0.000,B 0.000,C 90.000,E1 148.614} C_DIS
LIN {X -0.415,Y -642.426,Z 1167.620,A 0.000,B 0.000,C 90.000,E1 147.661} C_DIS
LIN {X -0.042,Y -644.331,Z 1167.615,A 0.000,B 0.000,C 90.000,E1 146.628} C_DIS
LIN {X -0.118,Y -646.646,Z 1167.608,A 0.000,B 0.000,C 90.000,E1 145.388} C_DIS
LIN {X 0.177,Y -649.729,Z 1167.598,A 0.000,B 0.000,C 90.000,E1 143.623} C_DIS
LIN {X 0.041,Y -651.864,Z 1167.591,A 0.000,B 0.000,C 90.000,E1 142.396} C_DIS
LIN {X -0.237,Y -657.233,Z 1167.575,A 0.000,B 0.000,C 90.000,E1 139.461} C_DIS
LIN {X 0.089,Y -660.781,Z 1167.565,A 0.000,B 0.000,C 90.000,E1 137.715} C_DIS
LIN {X 0.459,Y -664.335,Z 1167.556,A 0.000,B 0.000,C 90.000,E1 135.972} C_DIS
LIN {X -0.008,Y -669.544,Z 1167.542,A 0.000,B 0.000,C 90.000,E1 133.581} C_DIS
LIN {X -0.373,Y -673.577,Z 1167.533,A 0.000,B 0.000,C 90.000,E1 131.919} C_DIS
LIN {X -0.012,Y -679.367,Z 1167.519,A 0.000,B 0.000,C 90.000,E1 129.483} C_DIS
LIN {X -0.025,Y -683.535,Z 1167.510,A 0.000,B 0.000,C 90.000,E1 127.810} C_DIS
LIN {X 0.021,Y -687.100,Z 1167.502,A 0.000,B 0.000,C 90.000,E1 126.377} C_DIS
LIN {X 0.128,Y -690.646,Z 1167.494,A 0.000,B 0.000,C 90.000,E1 124.945} C_DIS
LIN {X -0.137,Y -693.430,Z 1167.488,A 0.000,B 0.000,C 90.000,E1 123.785} C_DIS
LIN {X -0.003,Y -695.595,Z 1167.482,A 0.000,B 0.000,C 90.000,E1 122.832} C_DIS
LIN {X 0.161,Y -697.647,Z 1167.477,A 0.000,B 0.000,C 90.000,E1 121.878} C_DIS
LIN {X 0.003,Y -699.916,Z 1167.471,A 0.000,B 0.000,C 90.000,E1 120.718} C_DIS
LIN {X -0.149,Y -701.609,Z 1167.465,A 0.000,B 0.000,C 90.000,E1 119.795} C_DIS
LIN {X 0.280,Y -704.046,Z 1167.458,A 0.000,B 0.000,C 90.000,E1 118.359} C_DIS
LIN {X -0.151,Y -705.483,Z 1167.453,A 0.000,B 0.000,C 90.000,E1 117.462} C_DIS
LIN {X 0.095,Y -706.160,Z 1167.449,A 0.000,B 0.000,C 90.000,E1 116.744} C_DIS
LIN {X -0.311,Y -706.643,Z 1167.443,A 0.000,B 0.000,C 90.000,E1 115.848} C_DIS
LIN {X -0.370,Y -706.748,Z 1167.440,A 0.000,B 0.000,C 90.000,E1 115.155} C_DIS
LIN {X 0.219,Y -706.475,Z 1167.437,A 0.000,B 0.000,C 90.000,E1 114.643} C_DIS
LIN {X -0.423,Y -706.222,Z 1167.436,A 0.000,B 0.000,C 90.000,E1 114.463} C_DIS
LIN {X 0.159,Y -705.332,Z 1167.433,A 0.000,B 0.000,C 90.000,E1 113.951} C_DIS
LIN {X 0.162,Y -704.429,Z 1167.432,A 0.000,B 0.000,C 90.000,E1 113.718} C_DIS
LIN {X 0.085,Y -702.221,Z 1167.429,A 0.000,B 0.000,C 90.000,E1 113.259} C_DIS
LIN {X -0.053,Y -701.275,Z 1167.429,A 0.000,B 0.000,C 90.000,E1 113.153} C_DIS
LIN {X -0.073,Y -696.704,Z 1167.426,A 0.000,B 0.000,C 90.000,E1 112.695} C_DIS
LIN {X -0.204,Y -694.971,Z 1167.425,A 0.000,B 0.000,C 90.000,E1 112.589} C_DIS
LIN {X 0.180,Y -692.460,Z 1167.425,A 0.000,B 0.000,C 90.000,E1 112.461} C_DIS
LIN {X -0.085,Y -685.888,Z 1167.424,A 0.000,B 0.000,C 90.000,E1 112.280} C_DIS
LIN {X -0.074,Y -684.898,Z 1167.424,A 0.000,B 0.000,C 90.000,E1 112.259} C_DIS
LIN {X -0.106,Y -676.366,Z 1167.423,A 0.000,B 0.000,C 90.000,E1 112.206} C_DIS
LIN {X -0.143,Y -604.673,Z 1167.423,A 0.000,B 0.000,C 90.000,E1 112.206} C_DIS
LIN {X -0.252,Y -599.895,Z 1167.422,A 0.000,B 0.000,C 90.000,E1 111.897} C_DIS
LIN {X 0.225,Y -595.751,Z 1167.420,A 0.000,B 0.000,C 90.000,E1 111.535} C_DIS
LIN {X 0.170,Y -581.356,Z 1167.413,A 0.000,B 0.000,C 90.000,E1 110.301} C_DIS
LIN {X 0.205,Y -574.261,Z 1167.410,A 0.000,B 0.000,C 90.000,E1 109.704} C_DIS
LIN {X -0.022,Y -568.337,Z 1167.407,A 0.000,B 0.000,C 90.000,E1 109.268} C_DIS
LIN {X 0.038,Y -560.438,Z 1167.404,A 0.000,B 0.000,C 90.000,E1 108.725} C_DIS
LIN {X 0.048,Y -555.781,Z 1167.402,A 0.000,B 0.000,C 90.000,E1 108.417} C_DIS
LIN {X 0.254,Y -551.736,Z 1167.401,A 0.000,B 0.000,C 90.000,E1 108.055} C_DIS
LIN {X -0.140,Y -550.422,Z 1167.399,A 0.000,B 0.000,C 90.000,E1 107.873} C_DIS
LIN {X -0.183,Y -550.405,Z 1167.399,A 0.000,B 0.000,C 90.000,E1 107.873} C_DIS
LIN {X -0.196,Y -549.970,Z 1167.397,A 0.000,B 0.000,C 90.000,E1 107.511} C_DIS
LIN {X 0.181,Y -550.378,Z 1167.393,A 0.000,B 0.000,C 90.000,E1 106.732} C_DIS
LIN {X 0.214,Y -551.341,Z 1167.387,A 0.000,B 0.000,C 90.000,E1 105.607} C_DIS
LIN {X 0.214,Y -553.000,Z 1167.376,A 0.000,B 0.000,C 90.000,E1 103.647} C_DIS
LIN {X -0.004,Y -554.786,Z 1167.365,A 0.000,B 0.000,C 90.000,E1 101.715} C_DIS
LIN {X 0.232,Y -556.469,Z 1167.356,A 0.000,B 0.000,C 90.000,E1 100.018} C_DIS
LIN {X 0.262,Y -557.825,Z 1167.348,A 0.000,B 0.000,C 90.000,E1 98.624} C_DIS
LIN {X 0.236,Y -559.086,Z 1167.340,A 0.000,B 0.000,C 90.000,E1 97.239} C_DIS
LIN {X -0.113,Y -560.534,Z 1167.330,A 0.000,B 0.000,C 90.000,E1 95.334} C_DIS
LIN {X -0.152,Y -561.473,Z 1167.322,A 0.000,B 0.000,C 90.000,E1 93.955} C_DIS
LIN {X -0.112,Y -562.681,Z 1167.313,A 0.000,B 0.000,C 90.000,E1 92.293} C_DIS
LIN {X 0.068,Y -564.182,Z 1167.302,A 0.000,B 0.000,C 90.000,E1 90.344} C_DIS
LIN {X -0.060,Y -564.943,Z 1167.296,A 0.000,B 0.000,C 90.000,E1 89.255} C_DIS
LIN {X -0.166,Y -565.666,Z 1167.290,A 0.000,B 0.000,C 90.000,E1 88.165} C_DIS
LIN {X 0.084,Y -566.859,Z 1167.279,A 0.000,B 0.000,C 90.000,E1 86.216} C_DIS
LIN {X -0.297,Y -567.881,Z 1167.270,A 0.000,B 0.000,C 90.000,E1 84.609} C_DIS
LIN {X 0.129,Y -569.185,Z 1167.259,A 0.000,B 0.000,C 90.000,E1 82.648} C_DIS
LIN {X -0.083,Y -570.101,Z 1167.250,A 0.000,B 0.000,C 90.000,E1 81.027} C_DIS
LIN {X -0.183,Y -570.937,Z 1167.241,A 0.000,B 0.000,C 90.000,E1 79.398} C_DIS
LIN {X 0.212,Y -571.610,Z 1167.234,A 0.000,B 0.000,C 90.000,E1 77.993} C_DIS
LIN {X 0.254,Y -572.410,Z 1167.224,A 0.000,B 0.000,C 90.000,E1 76.353} C_DIS
LIN {X 0.247,Y -573.108,Z 1167.217,A 0.000,B 0.000,C 90.000,E1 74.991} C_DIS
LIN {X 0.232,Y -574.450,Z 1167.203,A 0.000,B 0.000,C 90.000,E1 72.543} C_DIS
LIN {X 0.242,Y -575.871,Z 1167.191,A 0.000,B 0.000,C 90.000,E1 70.369} C_DIS
LIN {X 0.089,Y -576.920,Z 1167.184,A 0.000,B 0.000,C 90.000,E1 69.028} C_DIS
LIN {X -0.137,Y -578.624,Z 1167.173,A 0.000,B 0.000,C 90.000,E1 67.155} C_DIS
LIN {X -0.028,Y -579.995,Z 1167.166,A 0.000,B 0.000,C 90.000,E1 65.793} C_DIS
LIN {X 0.197,Y -581.459,Z 1167.157,A 0.000,B 0.000,C 90.000,E1 64.152} C_DIS
LIN {X 0.188,Y -583.002,Z 1167.148,A 0.000,B 0.000,C 90.000,E1 62.538} C_DIS
LIN {X 0.212,Y -584.478,Z 1167.139,A 0.000,B 0.000,C 90.000,E1 60.923} C_DIS
LIN {X 0.035,Y -585.867,Z 1167.130,A 0.000,B 0.000,C 90.000,E1 59.331} C_DIS
LIN {X -0.121,Y -587.053,Z 1167.121,A 0.000,B 0.000,C 90.000,E1 57.740} C_DIS
LIN {X -0.252,Y -588.379,Z 1167.110,A 0.000,B 0.000,C 90.000,E1 55.881} C_DIS
LIN {X -0.077,Y -589.220,Z 1167.103,A 0.000,B 0.000,C 90.000,E1 54.529} C_DIS
LIN {X 0.180,Y -590.372,Z 1167.093,A 0.000,B 0.000,C 90.000,E1 52.637} C_DIS
LIN {X 0.082,Y -591.602,Z 1167.081,A 0.000,B 0.000,C 90.000,E1 50.517} C_DIS
LIN {X -0.203,Y -591.946,Z 1167.076,A 0.000,B 0.000,C 90.000,E1 49.747} C_DIS
LIN {X -0.304,Y -592.389,Z 1167.068,A 0.000,B 0.000,C 90.000,E1 48.162} C_DIS
LIN {X -0.206,Y -592.579,Z 1167.060,A 0.000,B 0.000,C 90.000,E1 46.824} C_DIS
LIN {X 0.128,Y -592.539,Z 1167.054,A 0.000,B 0.000,C 90.000,E1 45.729} C_DIS
LIN {X -0.200,Y -592.216,Z 1167.047,A 0.000,B 0.000,C 90.000,E1 44.433} C_DIS
LIN {X -0.065,Y -591.899,Z 1167.042,A 0.000,B 0.000,C 90.000,E1 43.623} C_DIS
LIN {X 0.255,Y -591.338,Z 1167.036,A 0.000,B 0.000,C 90.000,E1 42.528} C_DIS
LIN {X 0.173,Y -590.599,Z 1167.031,A 0.000,B 0.000,C 90.000,E1 41.472} C_DIS
LIN {X -0.162,Y -589.340,Z 1167.023,A 0.000,B 0.000,C 90.000,E1 40.172} C_DIS
LIN {X -0.271,Y -588.136,Z 1167.017,A 0.000,B 0.000,C 90.000,E1 39.116} C_DIS
LIN {X 0.055,Y -586.755,Z 1167.011,A 0.000,B 0.000,C 90.000,E1 38.016} C_DIS
LIN {X 0.002,Y -585.123,Z 1167.005,A 0.000,B 0.000,C 90.000,E1 36.950} C_DIS
LIN {X -0.067,Y -583.196,Z 1166.999,A 0.000,B 0.000,C 90.000,E1 35.884} C_DIS
LIN {X -0.167,Y -580.733,Z 1166.993,A 0.000,B 0.000,C 90.000,E1 34.818} C_DIS
LIN {X -0.156,Y -579.411,Z 1166.990,A 0.000,B 0.000,C 90.000,E1 34.278} C_DIS
LIN {X 0.171,Y -577.837,Z 1166.987,A 0.000,B 0.000,C 90.000,E1 33.706} C_DIS
LIN {X 0.149,Y -574.440,Z 1166.981,A 0.000,B 0.000,C 90.000,E1 32.625} C_DIS
LIN {X 0.122,Y -572.470,Z 1166.978,A 0.000,B 0.000,C 90.000,E1 32.084} C_DIS
LIN {X 0.082,Y -570.269,Z 1166.975,A 0.000,B 0.000,C 90.000,E1 31.544} C_DIS
LIN {X 0.136,Y -566.642,Z 1166.971,A 0.000,B 0.000,C 90.000,E1 30.718} C_DIS
LIN {X -0.236,Y -564.063,Z 1166.968,A 0.000,B 0.000,C 90.000,E1 30.207} C_DIS
LIN {X 0.121,Y -559.032,Z 1166.962,A 0.000,B 0.000,C 90.000,E1 29.205} C_DIS
LIN {X 0.247,Y -554.245,Z 1166.958,A 0.000,B 0.000,C 90.000,E1 28.359} C_DIS
LIN {X -0.051,Y -550.007,Z 1166.954,A 0.000,B 0.000,C 90.000,E1 27.692} C_DIS
LIN {X -0.154,Y -545.425,Z 1166.950,A 0.000,B 0.000,C 90.000,E1 27.001} C_DIS
LIN {X 0.001,Y -540.395,Z 1166.946,A 0.000,B 0.000,C 90.000,E1 26.283} C_DIS
LIN {X -0.043,Y -536.019,Z 1166.943,A 0.000,B 0.000,C 90.000,E1 25.720} C_DIS
LIN {X -0.258,Y -530.220,Z 1166.939,A 0.000,B 0.000,C 90.000,E1 25.027} C_DIS
LIN {X 0.185,Y -524.143,Z 1166.935,A 0.000,B 0.000,C 90.000,E1 24.259} C_DIS
LIN {X 0.232,Y -516.310,Z 1166.930,A 0.000,B 0.000,C 90.000,E1 23.387} C_DIS
LIN {X 0.042,Y -509.583,Z 1166.926,A 0.000,B 0.000,C 90.000,E1 22.695} C_DIS
LIN {X -0.156,Y -502.694,Z 1166.922,A 0.000,B 0.000,C 90.000,E1 22.025} C_DIS
LIN {X 0.130,Y -492.797,Z 1166.917,A 0.000,B 0.000,C 90.000,E1 21.046} C_DIS
LIN {X 0.234,Y -481.388,Z 1166.911,A 0.000,B 0.000,C 90.000,E1 19.993} C_DIS
LIN {X 0.031,Y -469.573,Z 1166.905,A 0.000,B 0.000,C 90.000,E1 18.960} C_DIS
LIN {X 0.215,Y -457.694,Z 1166.900,A 0.000,B 0.000,C 90.000,E1 17.873} C_DIS
LIN {X -0.114,Y -446.185,Z 1166.894,A 0.000,B 0.000,C 90.000,E1 16.858} C_DIS
LIN {X -0.129,Y -428.823,Z 1166.884,A 0.000,B 0.000,C 90.000,E1 15.134} C_DIS
LIN {X -0.051,Y -413.436,Z 1166.875,A 0.000,B 0.000,C 90.000,E1 13.411} C_DIS
LIN {X 0.053,Y -405.559,Z 1166.869,A 0.000,B 0.000,C 90.000,E1 12.411} C_DIS
LIN {X 0.057,Y -398.051,Z 1166.863,A 0.000,B 0.000,C 90.000,E1 11.366} C_DIS
LIN {X 0.017,Y -395.275,Z 1166.861,A 0.000,B 0.000,C 90.000,E1 10.894} C_DIS
LIN {X -0.074,Y -393.186,Z 1166.858,A 0.000,B 0.000,C 90.000,E1 10.423} C_DIS
LIN {X -0.114,Y -392.633,Z 1166.856,A 0.000,B 0.000,C 90.000,E1 10.074} C_DIS
LIN {X -0.129,Y -393.504,Z 1166.853,A 0.000,B 0.000,C 90.000,E1 9.500} C_DIS
LIN {X 0.195,Y -396.000,Z 1166.848,A 0.000,B 0.000,C 90.000,E1 8.568} C_DIS
LIN {X 0.132,Y -398.447,Z 1166.844,A 0.000,B 0.000,C 90.000,E1 7.871} C_DIS
LIN {X 0.067,Y -401.824,Z 1166.839,A 0.000,B 0.000,C 90.000,E1 7.068} C_DIS
LIN {X 0.063,Y -404.276,Z 1166.837,A 0.000,B 0.000,C 90.000,E1 6.663} C_DIS
LIN {X 0.058,Y -406.471,Z 1166.835,A 0.000,B 0.000,C 90.000,E1 6.315} C_DIS
LIN {X 0.038,Y -407.828,Z 1166.834,A 0.000,B 0.000,C 90.000,E1 6.144} C_DIS
LIN {X 0.203,Y -411.093,Z 1166.832,A 0.000,B 0.000,C 90.000,E1 5.796} C_DIS
LIN {X 0.108,Y -426.523,Z 1166.826,A 0.000,B 0.000,C 90.000,E1 4.645} C_DIS
LIN {X -0.096,Y -445.678,Z 1166.818,A 0.000,B 0.000,C 90.000,E1 3.269} C_DIS
LIN {X 0.011,Y -463.532,Z 1166.811,A 0.000,B 0.000,C 90.000,E1 2.007} C_DIS
LIN {X 0.183,Y -473.030,Z 1166.807,A 0.000,B 0.000,C 90.000,E1 1.318} C_DIS
LIN {X 0.198,Y -482.452,Z 1166.804,A 0.000,B 0.000,C 90.000,E1 0.630} C_DIS
LIN {X 0.000,Y -490.917,Z 1166.800,A 0.000,B 0.000,C 90.000,E1 360.000} C_DIS
LIN {X 0.018,Y -496.419,Z 1166.797,A 0.000,B 0.000,C 90.000,E1 359.542} C_DIS
LIN {X 0.063,Y -503.324,Z 1166.794,A 0.000,B 0.000,C 90.000,E1 358.912} C_DIS
LIN {X 0.141,Y -510.140,Z 1166.790,A 0.000,B 0.000,C 90.000,E1 358.224} C_DIS
LIN {X 0.032,Y -516.646,Z 1166.786,A 0.000,B 0.000,C 90.000,E1 357.535} C_DIS
LIN {X 0.212,Y -522.831,Z 1166.782,A 0.000,B 0.000,C 90.000,E1 356.788} C_DIS
LIN {X 0.003,Y -528.354,Z 1166.778,A 0.000,B 0.000,C 90.000,E1 356.102} C_DIS
LIN {X -0.019,Y -532.508,Z 1166.775,A 0.000,B 0.000,C 90.000,E1 355.527} C_DIS
LIN {X 0.252,Y -537.194,Z 1166.771,A 0.000,B 0.000,C 90.000,E1 354.780} C_DIS
LIN {X 0.032,Y -541.376,Z 1166.767,A 0.000,B 0.000,C 90.000,E1 354.090} C_DIS
LIN {X -0.096,Y -545.097,Z 1166.763,A 0.000,B 0.000,C 90.000,E1 353.394} C_DIS
LIN {X 0.031,Y -549.254,Z 1166.759,A 0.000,B 0.000,C 90.000,E1 352.534} C_DIS
LIN {X 0.131,Y -550.591,Z 1166.757,A 0.000,B 0.000,C 90.000,E1 352.243} C_DIS
LIN {X -0.168,Y -554.017,Z 1166.752,A 0.000,B 0.000,C 90.000,E1 351.432} C_DIS
LIN {X 0.076,Y -556.124,Z 1166.749,A 0.000,B 0.000,C 90.000,E1 350.849} C_DIS
LIN {X -0.028,Y -559.898,Z 1166.743,A 0.000,B 0.000,C 90.000,E1 349.746} C_DIS
LIN {X 0.023,Y -563.201,Z 1166.737,A 0.000,B 0.000,C 90.000,E1 348.634} C_DIS
LIN {X 0.124,Y -566.237,Z 1166.731,A 0.000,B 0.000,C 90.000,E1 347.521} C_DIS
LIN {X -0.109,Y -569.763,Z 1166.723,A 0.000,B 0.000,C 90.000,E1 346.172} C_DIS
LIN {X -0.152,Y -573.003,Z 1166.716,A 0.000,B 0.000,C 90.000,E1 344.810} C_DIS
LIN {X 0.022,Y -574.819,Z 1166.711,A 0.000,B 0.000,C 90.000,E1 343.976} C_DIS
LIN {X -0.125,Y -578.340,Z 1166.702,A 0.000,B 0.000,C 90.000,E1 342.362} C_DIS
LIN {X 0.098,Y -579.984,Z 1166.698,A 0.000,B 0.000,C 90.000,E1 341.529} C_DIS
LIN {X -0.183,Y -582.047,Z 1166.692,A 0.000,B 0.000,C 90.000,E1 340.477} C_DIS
LIN {X -0.076,Y -583.849,Z 1166.686,A 0.000,B 0.000,C 90.000,E1 339.390} C_DIS
LIN {X 0.257,Y -585.382,Z 1166.680,A 0.000,B 0.000,C 90.000,E1 338.284} C_DIS
LIN {X 0.068,Y -586.578,Z 1166.674,A 0.000,B 0.000,C 90.000,E1 337.230} C_DIS
LIN {X 0.011,Y -587.201,Z 1166.669,A 0.000,B 0.000,C 90.000,E1 336.433} C_DIS
LIN {X 0.193,Y -587.564,Z 1166.665,A 0.000,B 0.000,C 90.000,E1 335.613} C_DIS
LIN {X 0.264,Y -587.513,Z 1166.659,A 0.000,B 0.000,C 90.000,E1 334.537} C_DIS
LIN {X -0.078,Y -587.124,Z 1166.654,A 0.000,B 0.000,C 90.000,E1 333.768} C_DIS
LIN {X -0.306,Y -586.662,Z 1166.651,A 0.000,B 0.000,C 90.000,E1 333.256} C_DIS
LIN {X 0.135,Y -585.685,Z 1166.647,A 0.000,B 0.000,C 90.000,E1 332.410} C_DIS
LIN {X -0.103,Y -584.812,Z 1166.644,A 0.000,B 0.000,C 90.000,E1 331.897} C_DIS
LIN {X 0.318,Y -583.233,Z 1166.639,A 0.000,B 0.000,C 90.000,E1 331.051} C_DIS
LIN {X 0.212,Y -581.215,Z 1166.635,A 0.000,B 0.000,C 90.000,E1 330.255} C_DIS
LIN {X 0.087,Y -578.769,Z 1166.630,A 0.000,B 0.000,C 90.000,E1 329.459} C_DIS
LIN {X -0.063,Y -575.608,Z 1166.626,A 0.000,B 0.000,C 90.000,E1 328.663} C_DIS
LIN {X -0.167,Y -572.228,Z 1166.622,A 0.000,B 0.000,C 90.000,E1 327.995} C_DIS
LIN {X 0.070,Y -566.850,Z 1166.617,A 0.000,B 0.000,C 90.000,E1 327.041} C_DIS
LIN {X -0.013,Y -563.184,Z 1166.614,A 0.000,B 0.000,C 90.000,E1 326.501} C_DIS
LIN {X -0.125,Y -559.194,Z 1166.611,A 0.000,B 0.000,C 90.000,E1 325.960} C_DIS
LIN {X -0.085,Y -555.318,Z 1166.608,A 0.000,B 0.000,C 90.000,E1 325.435} C_DIS
LIN {X -0.250,Y -550.688,Z 1166.605,A 0.000,B 0.000,C 90.000,E1 324.895} C_DIS
LIN {X -0.133,Y -545.835,Z 1166.602,A 0.000,B 0.000,C 90.000,E1 324.322} C_DIS
LIN {X -0.130,Y -533.619,Z 1166.594,A 0.000,B 0.000,C 90.000,E1 322.970} C_DIS
LIN {X -0.206,Y -527.341,Z 1166.590,A 0.000,B 0.000,C 90.000,E1 322.271} C_DIS
LIN {X -0.206,Y -524.442,Z 1166.588,A 0.000,B 0.000,C 90.000,E1 321.904} C_DIS
LIN {X -0.236,Y -522.369,Z 1166.587,A 0.000,B 0.000,C 90.000,E1 321.618} C_DIS
LIN {X -0.129,Y -520.146,Z 1166.584,A 0.000,B 0.000,C 90.000,E1 321.170} C_DIS
LIN {X -0.104,Y -518.203,Z 1166.581,A 0.000,B 0.000,C 90.000,E1 320.561} C_DIS
LIN {X -0.090,Y -517.276,Z 1166.577,A 0.000,B 0.000,C 90.000,E1 319.828} C_DIS
LIN {X 0.044,Y -517.287,Z 1166.572,A 0.000,B 0.000,C 90.000,E1 318.933} C_DIS
LIN {X -0.185,Y -518.350,Z 1166.561,A 0.000,B 0.000,C 90.000,E1 316.905} C_DIS
LIN {X 0.137,Y -519.121,Z 1166.552,A 0.000,B 0.000,C 90.000,E1 315.405} C_DIS
LIN {X 0.027,Y -520.050,Z 1166.543,A 0.000,B 0.000,C 90.000,E1 313.662} C_DIS
LIN {X 0.224,Y -521.196,Z 1166.531,A 0.000,B 0.000,C 90.000,E1 311.595} C_DIS
LIN {X 0.187,Y -522.249,Z 1166.522,A 0.000,B 0.000,C 90.000,E1 309.850} C_DIS
LIN {X 0.241,Y -523.289,Z 1166.512,A 0.000,B 0.000,C 90.000,E1 308.096} C_DIS
LIN {X 0.003,Y -524.356,Z 1166.502,A 0.000,B 0.000,C 90.000,E1 306.377} C_DIS
LIN {X 0.136,Y -525.654,Z 1166.489,A 0.000,B 0.000,C 90.000,E1 304.040} C_DIS
LIN {X -0.225,Y -526.764,Z 1166.480,A 0.000,B 0.000,C 90.000,E1 302.339} C_DIS
LIN {X -0.114,Y -527.764,Z 1166.470,A 0.000,B 0.000,C 90.000,E1 300.590} C_DIS
LIN {X 0.098,Y -528.310,Z 1166.464,A 0.000,B 0.000,C 90.000,E1 299.411} C_DIS
LIN {X 0.021,Y -528.853,Z 1166.455,A 0.000,B 0.000,C 90.000,E1 297.975} C_DIS
LIN {X 0.006,Y -529.124,Z 1166.449,A 0.000,B 0.000,C 90.000,E1 296.821} C_DIS
LIN {X -0.003,Y -529.310,Z 1166.443,A 0.000,B 0.000,C 90.000,E1 295.668} C_DIS
LIN {X 0.166,Y -529.360,Z 1166.435,A 0.000,B 0.000,C 90.000,E1 294.207} C_DIS
LIN {X -0.007,Y -529.300,Z 1166.423,A 0.000,B 0.000,C 90.000,E1 292.206} C_DIS
LIN {X -0.083,Y -529.058,Z 1166.414,A 0.000,B 0.000,C 90.000,E1 290.482} C_DIS
LIN {X 0.151,Y -528.634,Z 1166.404,A 0.000,B 0.000,C 90.000,E1 288.725} C_DIS
LIN {X 0.011,Y -528.342,Z 1166.399,A 0.000,B 0.000,C 90.000,E1 287.873} C_DIS
LIN {X 0.059,Y -527.699,Z 1166.390,A 0.000,B 0.000,C 90.000,E1 286.134} C_DIS
LIN {X -0.232,Y -527.164,Z 1166.383,A 0.000,B 0.000,C 90.000,E1 285.009} C_DIS
LIN {X 0.026,Y -526.150,Z 1166.374,A 0.000,B 0.000,C 90.000,E1 283.244} C_DIS
LIN {X 0.206,Y -525.661,Z 1166.369,A 0.000,B 0.000,C 90.000,E1 282.355} C_DIS
LIN {X -0.216,Y -524.705,Z 1166.361,A 0.000,B 0.000,C 90.000,E1 280.950} C_DIS
LIN {X -0.233,Y -523.730,Z 1166.353,A 0.000,B 0.000,C 90.000,E1 279.500} C_DIS
LIN {X -0.262,Y -522.790,Z 1166.345,A 0.000,B 0.000,C 90.000,E1 278.049} C_DIS
LIN {X 0.135,Y -521.744,Z 1166.335,A 0.000,B 0.000,C 90.000,E1 276.258} C_DIS
LIN {X -0.147,Y -520.514,Z 1166.322,A 0.000,B 0.000,C 90.000,E1 273.955} C_DIS
LIN {X 0.123,Y -519.864,Z 1166.314,A 0.000,B 0.000,C 90.000,E1 272.465} C_DIS
LIN {X -0.246,Y -518.983,Z 1166.302,A 0.000,B 0.000,C 90.000,E1 270.458} C_DIS
LIN {X -0.070,Y -518.232,Z 1166.293,A 0.000,B 0.000,C 90.000,E1 268.682} C_DIS
LIN {X 0.222,Y -517.652,Z 1166.286,A 0.000,B 0.000,C 90.000,E1 267.478} C_DIS
LIN {X -0.010,Y -517.004,Z 1166.280,A 0.000,B 0.000,C 90.000,E1 266.331} C_DIS
LIN {X -0.214,Y -516.185,Z 1166.273,A 0.000,B 0.000,C 90.000,E1 265.179} C_DIS
LIN {X 0.117,Y -515.514,Z 1166.268,A 0.000,B 0.000,C 90.000,E1 264.261} C_DIS
LIN {X -0.259,Y -513.577,Z 1166.257,A 0.000,B 0.000,C 90.000,E1 262.243} C_DIS
LIN {X 0.087,Y -512.694,Z 1166.252,A 0.000,B 0.000,C 90.000,E1 261.319} C_DIS
LIN {X -0.293,Y -510.195,Z 1166.237,A 0.000,B 0.000,C 90.000,E1 258.701} C_DIS
LIN {X 0.035,Y -508.407,Z 1166.226,A 0.000,B 0.000,C 90.000,E1 256.589} C_DIS
LIN {X -0.005,Y -506.917,Z 1166.216,A 0.000,B 0.000,C 90.000,E1 254.810} C_DIS
LIN {X -0.017,Y -505.622,Z 1166.207,A 0.000,B 0.000,C 90.000,E1 253.323} C_DIS
LIN {X 0.174,Y -503.971,Z 1166.197,A 0.000,B 0.000,C 90.000,E1 251.511} C_DIS
LIN {X -0.144,Y -502.320,Z 1166.188,A 0.000,B 0.000,C 90.000,E1 249.752} C_DIS
LIN {X -0.257,Y -500.349,Z 1166.176,A 0.000,B 0.000,C 90.000,E1 247.667} C_DIS
LIN {X -0.047,Y -499.446,Z 1166.171,A 0.000,B 0.000,C 90.000,E1 246.741} C_DIS
LIN {X 0.074,Y -497.243,Z 1166.161,A 0.000,B 0.000,C 90.000,E1 244.921} C_DIS
LIN {X -0.132,Y -495.289,Z 1166.152,A 0.000,B 0.000,C 90.000,E1 243.435} C_DIS
LIN {X 0.100,Y -492.844,Z 1166.142,A 0.000,B 0.000,C 90.000,E1 241.591} C_DIS
LIN {X -0.125,Y -490.282,Z 1166.132,A 0.000,B 0.000,C 90.000,E1 239.793} C_DIS
LIN {X 0.015,Y -487.663,Z 1166.122,A 0.000,B 0.000,C 90.000,E1 237.946} C_DIS
LIN {X 0.016,Y -484.418,Z 1166.110,A 0.000,B 0.000,C 90.000,E1 235.801} C_DIS
LIN {X 0.216,Y -481.297,Z 1166.098,A 0.000,B 0.000,C 90.000,E1 233.623} C_DIS
LIN {X -0.247,Y -478.544,Z 1166.088,A 0.000,B 0.000,C 90.000,E1 231.823} C_DIS
LIN {X -0.067,Y -476.721,Z 1166.081,A 0.000,B 0.000,C 90.000,E1 230.561} C_DIS
LIN {X -0.032,Y -474.175,Z 1166.071,A 0.000,B 0.000,C 90.000,E1 228.690} C_DIS
LIN {X -0.058,Y -472.768,Z 1166.065,A 0.000,B 0.000,C 90.000,E1 227.757} C_DIS
LIN {X 0.238,Y -467.360,Z 1166.046,A 0.000,B 0.000,C 90.000,E1 224.271} C_DIS
LIN {X 0.078,Y -464.790,Z 1166.034,A 0.000,B 0.000,C 90.000,E1 222.081} C_DIS
LIN {X 0.023,Y -461.888,Z 1166.009,A 0.000,B 0.000,C 90.000,E1 217.649} C_DIS
LIN {X 0.026,Y -460.917,Z 1165.995,A 0.000,B 0.000,C 90.000,E1 215.105} C_DIS
LIN {X 0.107,Y -460.769,Z 1165.976,A 0.000,B 0.000,C 90.000,E1 211.592} C_DIS
LIN {X -0.096,Y -462.403,Z 1165.958,A 0.000,B 0.000,C 90.000,E1 208.437} C_DIS
LIN {X -0.246,Y -466.489,Z 1165.935,A 0.000,B 0.000,C 90.000,E1 204.335} C_DIS
LIN {X -0.011,Y -472.322,Z 1165.916,A 0.000,B 0.000,C 90.000,E1 200.844} C_DIS
LIN {X -0.162,Y -478.741,Z 1165.900,A 0.000,B 0.000,C 90.000,E1 198.055} C_DIS
LIN {X -0.041,Y -488.549,Z 1165.881,A 0.000,B 0.000,C 90.000,E1 194.647} C_DIS
LIN {X 0.088,Y -492.515,Z 1165.875,A 0.000,B 0.000,C 90.000,E1 193.411} C_DIS
LIN {X 0.017,Y -499.618,Z 1165.863,A 0.000,B 0.000,C 90.000,E1 191.299} C_DIS
LIN {X -0.112,Y -508.020,Z 1165.849,A 0.000,B 0.000,C 90.000,E1 188.916} C_DIS
LIN {X 0.094,Y -513.447,Z 1165.841,A 0.000,B 0.000,C 90.000,E1 187.409} C_DIS
LIN {X -0.155,Y -517.729,Z 1165.835,A 0.000,B 0.000,C 90.000,E1 186.258} C_DIS
LIN {X 0.111,Y -524.045,Z 1165.825,A 0.000,B 0.000,C 90.000,E1 184.473} C_DIS
LIN {X -0.051,Y -530.383,Z 1165.815,A 0.000,B 0.000,C 90.000,E1 182.751} C_DIS
LIN {X -0.101,Y -535.590,Z 1165.807,A 0.000,B 0.000,C 90.000,E1 181.318} C_DIS
LIN {X -0.068,Y -540.809,Z 1165.799,A 0.000,B 0.000,C 90.000,E1 179.885} C_DIS
LIN {X 0.154,Y -548.121,Z 1165.788,A 0.000,B 0.000,C 90.000,E1 177.879} C_DIS
LIN {X -0.116,Y -553.253,Z 1165.781,A 0.000,B 0.000,C 90.000,E1 176.502} C_DIS
LIN {X -0.191,Y -559.426,Z 1165.771,A 0.000,B 0.000,C 90.000,E1 174.837} C_DIS
LIN {X -0.175,Y -564.526,Z 1165.764,A 0.000,B 0.000,C 90.000,E1 173.451} C_DIS
LIN {X 0.036,Y -570.636,Z 1165.754,A 0.000,B 0.000,C 90.000,E1 171.781} C_DIS
LIN {X -0.026,Y -576.653,Z 1165.745,A 0.000,B 0.000,C 90.000,E1 170.151} C_DIS
LIN {X -0.188,Y -581.560,Z 1165.738,A 0.000,B 0.000,C 90.000,E1 168.814} C_DIS
LIN {X 0.177,Y -585.459,Z 1165.732,A 0.000,B 0.000,C 90.000,E1 167.701} C_DIS
LIN {X -0.034,Y -591.090,Z 1165.723,A 0.000,B 0.000,C 90.000,E1 166.117} C_DIS
LIN {X -0.270,Y -595.653,Z 1165.716,A 0.000,B 0.000,C 90.000,E1 164.810} C_DIS
LIN {X 0.146,Y -600.116,Z 1165.708,A 0.000,B 0.000,C 90.000,E1 163.449} C_DIS
LIN {X 0.232,Y -604.338,Z 1165.701,A 0.000,B 0.000,C 90.000,E1 162.127} C_DIS
LIN {X 0.086,Y -607.607,Z 1165.695,A 0.000,B 0.000,C 90.000,E1 161.094} C_DIS
LIN {X -0.069,Y -611.535,Z 1165.688,A 0.000,B 0.000,C 90.000,E1 159.806} C_DIS
LIN {X -0.152,Y -615.349,Z 1165.681,A 0.000,B 0.000,C 90.000,E1 158.518} C_DIS
LIN {X -0.195,Y -619.595,Z 1165.672,A 0.000,B 0.000,C 90.000,E1 156.975} C_DIS
LIN {X 0.087,Y -623.151,Z 1165.665,A 0.000,B 0.000,C 90.000,E1 155.665} C_DIS
LIN {X -0.146,Y -626.548,Z 1165.658,A 0.000,B 0.000,C 90.000,E1 154.409} C_DIS
LIN {X -0.055,Y -629.844,Z 1165.651,A 0.000,B 0.000,C 90.000,E1 153.127} C_DIS
LIN {X 0.090,Y -633.023,Z 1165.644,A 0.000,B 0.000,C 90.000,E1 151.847} C_DIS
LIN {X -0.012,Y -635.434,Z 1165.638,A 0.000,B 0.000,C 90.000,E1 150.845} C_DIS
LIN {X -0.392,Y -637.779,Z 1165.632,A 0.000,B 0.000,C 90.000,E1 149.871} C_DIS
LIN {X -0.041,Y -640.538,Z 1165.625,A 0.000,B 0.000,C 90.000,E1 148.584} C_DIS
LIN {X 0.020,Y -643.039,Z 1165.619,A 0.000,B 0.000,C 90.000,E1 147.327} C_DIS
LIN {X 0.336,Y -645.860,Z 1165.610,A 0.000,B 0.000,C 90.000,E1 145.801} C_DIS
LIN {X 0.183,Y -648.487,Z 1165.602,A 0.000,B 0.000,C 90.000,E1 144.322} C_DIS
LIN {X 0.110,Y -650.224,Z 1165.596,A 0.000,B 0.000,C 90.000,E1 143.336} C_DIS
LIN {X -0.018,Y -652.304,Z 1165.590,A 0.000,B 0.000,C 90.000,E1 142.110} C_DIS
LIN {X 0.225,Y -656.804,Z 1165.576,A 0.000,B 0.000,C 90.000,E1 139.622} C_DIS
LIN {X 0.050,Y -660.338,Z 1165.566,A 0.000,B 0.000,C 90.000,E1 137.919} C_DIS
LIN {X -0.040,Y -663.911,Z 1165.557,A 0.000,B 0.000,C 90.000,E1 136.215} C_DIS
LIN {X -0.057,Y -669.601,Z 1165.542,A 0.000,B 0.000,C 90.000,E1 133.542} C_DIS
LIN {X 0.064,Y -673.622,Z 1165.532,A 0.000,B 0.000,C 90.000,E1 131.838} C_DIS
LIN {X 0.403,Y -678.807,Z 1165.521,A 0.000,B 0.000,C 90.000,E1 129.644} C_DIS
LIN {X 0.212,Y -681.779,Z 1165.514,A 0.000,B 0.000,C 90.000,E1 128.463} C_DIS
LIN {X 0.417,Y -683.595,Z 1165.510,A 0.000,B 0.000,C 90.000,E1 127.729} C_DIS
LIN {X -0.091,Y -687.163,Z 1165.502,A 0.000,B 0.000,C 90.000,E1 126.343} C_DIS
LIN {X 0.174,Y -690.706,Z 1165.494,A 0.000,B 0.000,C 90.000,E1 124.898} C_DIS
LIN {X -0.052,Y -694.065,Z 1165.486,A 0.000,B 0.000,C 90.000,E1 123.499} C_DIS
LIN {X -0.260,Y -696.694,Z 1165.480,A 0.000,B 0.000,C 90.000,E1 122.339} C_DIS
LIN {X -0.091,Y -698.629,Z 1165.474,A 0.000,B 0.000,C 90.000,E1 121.386} C_DIS
LIN {X 0.005,Y -700.818,Z 1165.468,A 0.000,B 0.000,C 90.000,E1 120.207} C_DIS
LIN {X 0.091,Y -703.712,Z 1165.459,A 0.000,B 0.000,C 90.000,E1 118.565} C_DIS
LIN {X -0.300,Y -704.857,Z 1165.455,A 0.000,B 0.000,C 90.000,E1 117.897} C_DIS
LIN {X 0.275,Y -705.515,Z 1165.452,A 0.000,B 0.000,C 90.000,E1 117.385} C_DIS
LIN {X 0.200,Y -706.175,Z 1165.448,A 0.000,B 0.000,C 90.000,E1 116.693} C_DIS
LIN {X -0.200,Y -706.654,Z 1165.443,A 0.000,B 0.000,C 90.000,E1 115.796} C_DIS
LIN {X 0.045,Y -706.725,Z 1165.439,A 0.000,B 0.000,C 90.000,E1 115.079} C_DIS
LIN {X -0.306,Y -706.448,Z 1165.437,A 0.000,B 0.000,C 90.000,E1 114.643} C_DIS
LIN {X -0.013,Y -705.684,Z 1165.434,A 0.000,B 0.000,C 90.000,E1 114.155} C_DIS
LIN {X 0.279,Y -705.223,Z 1165.433,A 0.000,B 0.000,C 90.000,E1 113.898} C_DIS
LIN {X 0.065,Y -702.650,Z 1165.430,A 0.000,B 0.000,C 90.000,E1 113.334} C_DIS
LIN {X 0.205,Y -701.917,Z 1165.429,A 0.000,B 0.000,C 90.000,E1 113.206} C_DIS
LIN {X -0.170,Y -697.439,Z 1165.427,A 0.000,B 0.000,C 90.000,E1 112.770} C_DIS
LIN {X -0.034,Y -696.094,Z 1165.426,A 0.000,B 0.000,C 90.000,E1 112.642} C_DIS
LIN {X 0.100,Y -693.912,Z 1165.425,A 0.000,B 0.000,C 90.000,E1 112.514} C_DIS
LIN {X -0.360,Y -686.970,Z 1165.424,A 0.000,B 0.000,C 90.000,E1 112.333} C_DIS
LIN {X -0.105,Y -684.935,Z 1165.424,A 0.000,B 0.000,C 90.000,E1 112.259} C_DIS
LIN {X -0.131,Y -677.165,Z 1165.423,A 0.000,B 0.000,C 90.000,E1 112.206} C_DIS
LIN {X -0.165,Y -604.562,Z 1165.423,A 0.000,B 0.000,C 90.000,E1 112.206} C_DIS
LIN {X 0.204,Y -599.694,Z 1165.422,A 0.000,B 0.000,C 90.000,E1 111.844} C_DIS
LIN {X 0.123,Y -595.565,Z 1165.420,A 0.000,B 0.000,C 90.000,E1 111.535} C_DIS
LIN {X 0.123,Y -579.831,Z 1165.412,A 0.000,B 0.000,C 90.000,E1 110.174} C_DIS
LIN {X 0.057,Y -574.101,Z 1165.410,A 0.000,B 0.000,C 90.000,E1 109.704} C_DIS
LIN {X -0.151,Y -568.194,Z 1165.407,A 0.000,B 0.000,C 90.000,E1 109.268} C_DIS
LIN {X -0.083,Y -560.293,Z 1165.404,A 0.000,B 0.000,C 90.000,E1 108.725} C_DIS
LIN {X -0.071,Y -555.618,Z 1165.402,A 0.000,B 0.000,C 90.000,E1 108.417} C_DIS
LIN {X 0.147,Y -551.599,Z 1165.400,A 0.000,B 0.000,C 90.000,E1 108.055} C_DIS
LIN {X -0.078,Y -550.390,Z 1165.399,A 0.000,B 0.000,C 90.000,E1 107.873} C_DIS
LIN {X -0.120,Y -550.373,Z 1165.399,A 0.000,B 0.000,C 90.000,E1 107.873} C_DIS
LIN {X 0.223,Y -549.955,Z 1165.397,A 0.000,B 0.000,C 90.000,E1 107.457} C_DIS
LIN {X 0.073,Y -550.367,Z 1165.393,A 0.000,B 0.000,C 90.000,E1 106.732} C_DIS
LIN {X 0.107,Y -551.324,Z 1165.387,A 0.000,B 0.000,C 90.000,E1 105.607} C_DIS
LIN {X 0.106,Y -552.960,Z 1165.376,A 0.000,B 0.000,C 90.000,E1 103.647} C_DIS
LIN {X -0.114,Y -554.737,Z 1165.365,A 0.000,B 0.000,C 90.000,E1 101.715} C_DIS
LIN {X -0.010,Y -556.172,Z 1165.357,A 0.000,B 0.000,C 90.000,E1 100.310} C_DIS
LIN {X 0.150,Y -557.767,Z 1165.348,A 0.000,B 0.000,C 90.000,E1 98.624} C_DIS
LIN {X 0.122,Y -559.004,Z 1165.340,A 0.000,B 0.000,C 90.000,E1 97.239} C_DIS
LIN {X -0.229,Y -560.451,Z 1165.330,A 0.000,B 0.000,C 90.000,E1 95.334} C_DIS
LIN {X 0.290,Y -561.410,Z 1165.322,A 0.000,B 0.000,C 90.000,E1 93.898} C_DIS
LIN {X -0.231,Y -562.627,Z 1165.313,A 0.000,B 0.000,C 90.000,E1 92.293} C_DIS
LIN {X -0.159,Y -563.886,Z 1165.303,A 0.000,B 0.000,C 90.000,E1 90.630} C_DIS
LIN {X 0.163,Y -564.532,Z 1165.299,A 0.000,B 0.000,C 90.000,E1 89.771} C_DIS
LIN {X 0.277,Y -565.605,Z 1165.290,A 0.000,B 0.000,C 90.000,E1 88.108} C_DIS
LIN {X -0.041,Y -566.788,Z 1165.279,A 0.000,B 0.000,C 90.000,E1 86.216} C_DIS
LIN {X 0.141,Y -567.776,Z 1165.270,A 0.000,B 0.000,C 90.000,E1 84.552} C_DIS
LIN {X -0.001,Y -569.076,Z 1165.259,A 0.000,B 0.000,C 90.000,E1 82.648} C_DIS
LIN {X -0.215,Y -569.994,Z 1165.250,A 0.000,B 0.000,C 90.000,E1 81.027} C_DIS
LIN {X 0.242,Y -570.806,Z 1165.241,A 0.000,B 0.000,C 90.000,E1 79.342} C_DIS
LIN {X 0.075,Y -571.471,Z 1165.233,A 0.000,B 0.000,C 90.000,E1 77.993} C_DIS
LIN {X -0.252,Y -572.411,Z 1165.223,A 0.000,B 0.000,C 90.000,E1 76.117} C_DIS
LIN {X 0.084,Y -573.201,Z 1165.214,A 0.000,B 0.000,C 90.000,E1 74.448} C_DIS
LIN {X -0.280,Y -574.493,Z 1165.202,A 0.000,B 0.000,C 90.000,E1 72.308} C_DIS
LIN {X 0.093,Y -576.183,Z 1165.188,A 0.000,B 0.000,C 90.000,E1 69.826} C_DIS
LIN {X 0.004,Y -578.017,Z 1165.176,A 0.000,B 0.000,C 90.000,E1 67.667} C_DIS
LIN {X -0.048,Y -579.630,Z 1165.167,A 0.000,B 0.000,C 90.000,E1 66.049} C_DIS
LIN {X 0.168,Y -581.107,Z 1165.158,A 0.000,B 0.000,C 90.000,E1 64.409} C_DIS
LIN {X 0.020,Y -582.881,Z 1165.147,A 0.000,B 0.000,C 90.000,E1 62.538} C_DIS
LIN {X 0.041,Y -584.359,Z 1165.139,A 0.000,B 0.000,C 90.000,E1 60.923} C_DIS
LIN {X -0.139,Y -585.710,Z 1165.130,A 0.000,B 0.000,C 90.000,E1 59.331} C_DIS
LIN {X -0.168,Y -586.724,Z 1165.122,A 0.000,B 0.000,C 90.000,E1 57.995} C_DIS
LIN {X 0.189,Y -588.052,Z 1165.112,A 0.000,B 0.000,C 90.000,E1 56.087} C_DIS
LIN {X 0.218,Y -589.027,Z 1165.103,A 0.000,B 0.000,C 90.000,E1 54.482} C_DIS
LIN {X -0.010,Y -590.195,Z 1165.093,A 0.000,B 0.000,C 90.000,E1 52.637} C_DIS
LIN {X -0.113,Y -591.404,Z 1165.081,A 0.000,B 0.000,C 90.000,E1 50.517} C_DIS
LIN {X -0.193,Y -591.826,Z 1165.075,A 0.000,B 0.000,C 90.000,E1 49.461} C_DIS
LIN {X 0.331,Y -592.166,Z 1165.067,A 0.000,B 0.000,C 90.000,E1 48.081} C_DIS
LIN {X -0.177,Y -592.322,Z 1165.061,A 0.000,B 0.000,C 90.000,E1 47.067} C_DIS
LIN {X 0.152,Y -592.305,Z 1165.056,A 0.000,B 0.000,C 90.000,E1 45.972} C_DIS
LIN {X 0.055,Y -592.114,Z 1165.050,A 0.000,B 0.000,C 90.000,E1 44.919} C_DIS
LIN {X -0.046,Y -591.753,Z 1165.044,A 0.000,B 0.000,C 90.000,E1 43.866} C_DIS
LIN {X 0.035,Y -591.075,Z 1165.036,A 0.000,B 0.000,C 90.000,E1 42.528} C_DIS
LIN {X -0.051,Y -590.301,Z 1165.030,A 0.000,B 0.000,C 90.000,E1 41.472} C_DIS
LIN {X -0.011,Y -588.991,Z 1165.023,A 0.000,B 0.000,C 90.000,E1 40.135} C_DIS
LIN {X -0.308,Y -587.446,Z 1165.016,A 0.000,B 0.000,C 90.000,E1 38.830} C_DIS
LIN {X -0.184,Y -586.385,Z 1165.011,A 0.000,B 0.000,C 90.000,E1 38.016} C_DIS
LIN {X -0.240,Y -584.700,Z 1165.005,A 0.000,B 0.000,C 90.000,E1 36.950} C_DIS
LIN {X -0.153,Y -583.266,Z 1165.001,A 0.000,B 0.000,C 90.000,E1 36.137} C_DIS
LIN {X 0.044,Y -581.563,Z 1164.996,A 0.000,B 0.000,C 90.000,E1 35.311} C_DIS
LIN {X -0.085,Y -578.874,Z 1164.990,A 0.000,B 0.000,C 90.000,E1 34.246} C_DIS
LIN {X -0.087,Y -577.298,Z 1164.987,A 0.000,B 0.000,C 90.000,E1 33.706} C_DIS
LIN {X -0.116,Y -573.834,Z 1164.981,A 0.000,B 0.000,C 90.000,E1 32.625} C_DIS
LIN {X -0.016,Y -570.738,Z 1164.977,A 0.000,B 0.000,C 90.000,E1 31.799} C_DIS
LIN {X -0.069,Y -568.433,Z 1164.974,A 0.000,B 0.000,C 90.000,E1 31.258} C_DIS
LIN {X 0.161,Y -564.681,Z 1164.969,A 0.000,B 0.000,C 90.000,E1 30.413} C_DIS
LIN {X -0.136,Y -560.464,Z 1164.964,A 0.000,B 0.000,C 90.000,E1 29.617} C_DIS
LIN {X -0.267,Y -557.479,Z 1164.961,A 0.000,B 0.000,C 90.000,E1 29.077} C_DIS
LIN {X -0.045,Y -553.459,Z 1164.958,A 0.000,B 0.000,C 90.000,E1 28.359} C_DIS
LIN {X 0.253,Y -550.068,Z 1164.954,A 0.000,B 0.000,C 90.000,E1 27.769} C_DIS
LIN {X -0.214,Y -546.458,Z 1164.951,A 0.000,B 0.000,C 90.000,E1 27.257} C_DIS
LIN {X -0.091,Y -543.567,Z 1164.949,A 0.000,B 0.000,C 90.000,E1 26.821} C_DIS
LIN {X 0.130,Y -539.410,Z 1164.946,A 0.000,B 0.000,C 90.000,E1 26.232} C_DIS
LIN {X -0.059,Y -533.860,Z 1164.942,A 0.000,B 0.000,C 90.000,E1 25.540} C_DIS
LIN {X 0.274,Y -526.808,Z 1164.937,A 0.000,B 0.000,C 90.000,E1 24.643} C_DIS
LIN {X 0.141,Y -521.750,Z 1164.934,A 0.000,B 0.000,C 90.000,E1 24.079} C_DIS
LIN {X 0.122,Y -515.441,Z 1164.930,A 0.000,B 0.000,C 90.000,E1 23.387} C_DIS
LIN {X -0.016,Y -508.743,Z 1164.926,A 0.000,B 0.000,C 90.000,E1 22.695} C_DIS
LIN {X -0.236,Y -501.819,Z 1164.922,A 0.000,B 0.000,C 90.000,E1 22.025} C_DIS
LIN {X 0.180,Y -492.059,Z 1164.917,A 0.000,B 0.000,C 90.000,E1 21.046} C_DIS
LIN {X 0.123,Y -480.375,Z 1164.911,A 0.000,B 0.000,C 90.000,E1 19.993} C_DIS
LIN {X -0.088,Y -467.172,Z 1164.905,A 0.000,B 0.000,C 90.000,E1 18.833} C_DIS
LIN {X -0.119,Y -452.328,Z 1164.897,A 0.000,B 0.000,C 90.000,E1 17.511} C_DIS
LIN {X 0.158,Y -430.693,Z 1164.886,A 0.000,B 0.000,C 90.000,E1 15.371} C_DIS
LIN {X -0.097,Y -415.228,Z 1164.876,A 0.000,B 0.000,C 90.000,E1 13.703} C_DIS
LIN {X -0.015,Y -407.151,Z 1164.871,A 0.000,B 0.000,C 90.000,E1 12.703} C_DIS
LIN {X 0.007,Y -399.458,Z 1164.865,A 0.000,B 0.000,C 90.000,E1 11.658} C_DIS
LIN {X 0.053,Y -395.215,Z 1164.861,A 0.000,B 0.000,C 90.000,E1 10.950} C_DIS
LIN {X -0.128,Y -393.155,Z 1164.858,A 0.000,B 0.000,C 90.000,E1 10.489} C_DIS
LIN {X -0.166,Y -392.591,Z 1164.856,A 0.000,B 0.000,C 90.000,E1 10.141} C_DIS
LIN {X 0.025,Y -393.177,Z 1164.854,A 0.000,B 0.000,C 90.000,E1 9.670} C_DIS
LIN {X -0.018,Y -393.998,Z 1164.852,A 0.000,B 0.000,C 90.000,E1 9.321} C_DIS
LIN {X -0.142,Y -396.606,Z 1164.847,A 0.000,B 0.000,C 90.000,E1 8.454} C_DIS
LIN {X -0.215,Y -398.427,Z 1164.844,A 0.000,B 0.000,C 90.000,E1 7.936} C_DIS
LIN {X -0.121,Y -401.896,Z 1164.839,A 0.000,B 0.000,C 90.000,E1 7.068} C_DIS
LIN {X -0.103,Y -402.825,Z 1164.838,A 0.000,B 0.000,C 90.000,E1 6.891} C_DIS
LIN {X -0.097,Y -406.746,Z 1164.835,A 0.000,B 0.000,C 90.000,E1 6.258} C_DIS
LIN {X 0.042,Y -409.744,Z 1164.833,A 0.000,B 0.000,C 90.000,E1 5.910} C_DIS
LIN {X 0.186,Y -411.237,Z 1164.832,A 0.000,B 0.000,C 90.000,E1 5.739} C_DIS
LIN {X 0.206,Y -424.963,Z 1164.826,A 0.000,B 0.000,C 90.000,E1 4.702} C_DIS
LIN {X -0.081,Y -441.117,Z 1164.820,A 0.000,B 0.000,C 90.000,E1 3.555} C_DIS
LIN {X 0.069,Y -463.753,Z 1164.811,A 0.000,B 0.000,C 90.000,E1 1.949} C_DIS
LIN {X -0.217,Y -473.229,Z 1164.807,A 0.000,B 0.000,C 90.000,E1 1.318} C_DIS
LIN {X -0.209,Y -482.675,Z 1164.803,A 0.000,B 0.000,C 90.000,E1 0.630} C_DIS
LIN {X 0.000,Y -490.599,Z 1164.800,A 0.000,B 0.000,C 90.000,E1 360.000} C_DIS
LIN {X -0.061,Y -497.523,Z 1164.797,A 0.000,B 0.000,C 90.000,E1 359.427} C_DIS
LIN {X -0.056,Y -503.248,Z 1164.794,A 0.000,B 0.000,C 90.000,E1 358.912} C_DIS
LIN {X 0.026,Y -510.129,Z 1164.790,A 0.000,B 0.000,C 90.000,E1 358.224} C_DIS
LIN {X 0.034,Y -516.573,Z 1164.786,A 0.000,B 0.000,C 90.000,E1 357.535} C_DIS
LIN {X -0.247,Y -522.768,Z 1164.782,A 0.000,B 0.000,C 90.000,E1 356.846} C_DIS
LIN {X -0.100,Y -528.504,Z 1164.778,A 0.000,B 0.000,C 90.000,E1 356.102} C_DIS
LIN {X -0.122,Y -532.678,Z 1164.775,A 0.000,B 0.000,C 90.000,E1 355.527} C_DIS
LIN {X 0.151,Y -537.369,Z 1164.771,A 0.000,B 0.000,C 90.000,E1 354.780} C_DIS
LIN {X -0.069,Y -541.602,Z 1164.767,A 0.000,B 0.000,C 90.000,E1 354.090} C_DIS
LIN {X -0.196,Y -545.364,Z 1164.763,A 0.000,B 0.000,C 90.000,E1 353.394} C_DIS
LIN {X -0.091,Y -548.163,Z 1164.760,A 0.000,B 0.000,C 90.000,E1 352.818} C_DIS
LIN {X -0.225,Y -551.456,Z 1164.756,A 0.000,B 0.000,C 90.000,E1 352.129} C_DIS
LIN {X -0.260,Y -554.316,Z 1164.752,A 0.000,B 0.000,C 90.000,E1 351.432} C_DIS
LIN {X -0.015,Y -556.416,Z 1164.749,A 0.000,B 0.000,C 90.000,E1 350.849} C_DIS
LIN {X -0.114,Y -560.217,Z 1164.743,A 0.000,B 0.000,C 90.000,E1 349.746} C_DIS
LIN {X -0.060,Y -563.551,Z 1164.737,A 0.000,B 0.000,C 90.000,E1 348.634} C_DIS
LIN {X 0.218,Y -567.336,Z 1164.729,A 0.000,B 0.000,C 90.000,E1 347.229} C_DIS
LIN {X 0.000,Y -570.783,Z 1164.722,A 0.000,B 0.000,C 90.000,E1 345.880} C_DIS
LIN {X -0.218,Y -573.401,Z 1164.716,A 0.000,B 0.000,C 90.000,E1 344.810} C_DIS
LIN {X 0.154,Y -575.820,Z 1164.709,A 0.000,B 0.000,C 90.000,E1 343.685} C_DIS
LIN {X 0.199,Y -579.362,Z 1164.700,A 0.000,B 0.000,C 90.000,E1 342.054} C_DIS
LIN {X -0.116,Y -580.977,Z 1164.696,A 0.000,B 0.000,C 90.000,E1 341.275} C_DIS
LIN {X -0.023,Y -583.006,Z 1164.690,A 0.000,B 0.000,C 90.000,E1 340.188} C_DIS
LIN {X -0.051,Y -585.148,Z 1164.682,A 0.000,B 0.000,C 90.000,E1 338.847} C_DIS
LIN {X 0.228,Y -585.924,Z 1164.680,A 0.000,B 0.000,C 90.000,E1 338.284} C_DIS
LIN {X -0.075,Y -587.374,Z 1164.672,A 0.000,B 0.000,C 90.000,E1 336.975} C_DIS
LIN {X -0.124,Y -587.906,Z 1164.668,A 0.000,B 0.000,C 90.000,E1 336.177} C_DIS
LIN {X 0.067,Y -588.168,Z 1164.663,A 0.000,B 0.000,C 90.000,E1 335.357} C_DIS
LIN {X 0.262,Y -588.134,Z 1164.659,A 0.000,B 0.000,C 90.000,E1 334.537} C_DIS
LIN {X -0.075,Y -587.825,Z 1164.654,A 0.000,B 0.000,C 90.000,E1 333.768} C_DIS
LIN {X 0.111,Y -587.072,Z 1164.650,A 0.000,B 0.000,C 90.000,E1 332.948} C_DIS
LIN {X 0.035,Y -586.061,Z 1164.645,A 0.000,B 0.000,C 90.000,E1 332.153} C_DIS
LIN {X 0.347,Y -583.995,Z 1164.639,A 0.000,B 0.000,C 90.000,E1 331.051} C_DIS
LIN {X 0.248,Y -582.015,Z 1164.635,A 0.000,B 0.000,C 90.000,E1 330.255} C_DIS
LIN {X -0.022,Y -580.423,Z 1164.632,A 0.000,B 0.000,C 90.000,E1 329.744} C_DIS
LIN {X -0.011,Y -578.611,Z 1164.629,A 0.000,B 0.000,C 90.000,E1 329.203} C_DIS
LIN {X -0.010,Y -576.521,Z 1164.626,A 0.000,B 0.000,C 90.000,E1 328.663} C_DIS
LIN {X 0.058,Y -574.602,Z 1164.624,A 0.000,B 0.000,C 90.000,E1 328.250} C_DIS
LIN {X 0.031,Y -571.732,Z 1164.621,A 0.000,B 0.000,C 90.000,E1 327.709} C_DIS
LIN {X -0.018,Y -568.686,Z 1164.618,A 0.000,B 0.000,C 90.000,E1 327.168} C_DIS
LIN {X -0.187,Y -564.151,Z 1164.614,A 0.000,B 0.000,C 90.000,E1 326.501} C_DIS
LIN {X -0.087,Y -559.232,Z 1164.610,A 0.000,B 0.000,C 90.000,E1 325.801} C_DIS
LIN {X -0.109,Y -556.128,Z 1164.608,A 0.000,B 0.000,C 90.000,E1 325.388} C_DIS
LIN {X -0.207,Y -549.099,Z 1164.603,A 0.000,B 0.000,C 90.000,E1 324.562} C_DIS
LIN {X 0.083,Y -542.931,Z 1164.599,A 0.000,B 0.000,C 90.000,E1 323.829} C_DIS
LIN {X -0.184,Y -532.896,Z 1164.593,A 0.000,B 0.000,C 90.000,E1 322.763} C_DIS
LIN {X 0.050,Y -526.640,Z 1164.589,A 0.000,B 0.000,C 90.000,E1 322.029} C_DIS
LIN {X 0.046,Y -523.864,Z 1164.587,A 0.000,B 0.000,C 90.000,E1 321.662} C_DIS
LIN {X 0.114,Y -521.120,Z 1164.584,A 0.000,B 0.000,C 90.000,E1 321.170} C_DIS
LIN {X -0.154,Y -519.883,Z 1164.583,A 0.000,B 0.000,C 90.000,E1 320.884} C_DIS
LIN {X 0.122,Y -518.856,Z 1164.581,A 0.000,B 0.000,C 90.000,E1 320.561} C_DIS
LIN {X 0.142,Y -517.720,Z 1164.577,A 0.000,B 0.000,C 90.000,E1 319.828} C_DIS
LIN {X 0.163,Y -517.775,Z 1164.570,A 0.000,B 0.000,C 90.000,E1 318.609} C_DIS
LIN {X 0.049,Y -518.677,Z 1164.560,A 0.000,B 0.000,C 90.000,E1 316.863} C_DIS
LIN {X -0.002,Y -519.407,Z 1164.552,A 0.000,B 0.000,C 90.000,E1 315.405} C_DIS
LIN {X 0.253,Y -520.327,Z 1164.543,A 0.000,B 0.000,C 90.000,E1 313.623} C_DIS
LIN {X 0.098,Y -521.448,Z 1164.531,A 0.000,B 0.000,C 90.000,E1 311.595} C_DIS
LIN {X -0.221,Y -522.319,Z 1164.523,A 0.000,B 0.000,C 90.000,E1 310.172} C_DIS
LIN {X 0.125,Y -523.511,Z 1164.512,A 0.000,B 0.000,C 90.000,E1 308.096} C_DIS
LIN {X -0.109,Y -524.590,Z 1164.502,A 0.000,B 0.000,C 90.000,E1 306.377} C_DIS
LIN {X 0.067,Y -525.714,Z 1164.491,A 0.000,B 0.000,C 90.000,E1 304.326} C_DIS
LIN {X 0.120,Y -527.003,Z 1164.479,A 0.000,B 0.000,C 90.000,E1 302.291} C_DIS
LIN {X -0.209,Y -528.033,Z 1164.470,A 0.000,B 0.000,C 90.000,E1 300.590} C_DIS
LIN {X 0.312,Y -528.517,Z 1164.465,A 0.000,B 0.000,C 90.000,E1 299.667} C_DIS
LIN {X -0.065,Y -529.204,Z 1164.455,A 0.000,B 0.000,C 90.000,E1 297.975} C_DIS
LIN {X -0.248,Y -529.439,Z 1164.451,A 0.000,B 0.000,C 90.000,E1 297.129} C_DIS
LIN {X -0.078,Y -529.682,Z 1164.443,A 0.000,B 0.000,C 90.000,E1 295.668} C_DIS
LIN {X 0.098,Y -529.719,Z 1164.435,A 0.000,B 0.000,C 90.000,E1 294.207} C_DIS
LIN {X -0.066,Y -529.658,Z 1164.423,A 0.000,B 0.000,C 90.000,E1 292.206} C_DIS
LIN {X 0.177,Y -529.521,Z 1164.415,A 0.000,B 0.000,C 90.000,E1 290.737} C_DIS
LIN {X 0.108,Y -529.003,Z 1164.404,A 0.000,B 0.000,C 90.000,E1 288.725} C_DIS
LIN {X -0.013,Y -528.578,Z 1164.398,A 0.000,B 0.000,C 90.000,E1 287.583} C_DIS
LIN {X 0.028,Y -528.029,Z 1164.390,A 0.000,B 0.000,C 90.000,E1 286.134} C_DIS
LIN {X 0.253,Y -527.515,Z 1164.383,A 0.000,B 0.000,C 90.000,E1 284.954} C_DIS
LIN {X 0.009,Y -526.531,Z 1164.374,A 0.000,B 0.000,C 90.000,E1 283.244} C_DIS
LIN {X 0.213,Y -525.820,Z 1164.367,A 0.000,B 0.000,C 90.000,E1 282.063} C_DIS
LIN {X -0.224,Y -525.082,Z 1164.361,A 0.000,B 0.000,C 90.000,E1 280.950} C_DIS
LIN {X -0.233,Y -524.097,Z 1164.353,A 0.000,B 0.000,C 90.000,E1 279.500} C_DIS
LIN {X -0.250,Y -522.987,Z 1164.343,A 0.000,B 0.000,C 90.000,E1 277.757} C_DIS
LIN {X 0.146,Y -521.940,Z 1164.333,A 0.000,B 0.000,C 90.000,E1 275.967} C_DIS
LIN {X -0.121,Y -520.923,Z 1164.322,A 0.000,B 0.000,C 90.000,E1 273.955} C_DIS
LIN {X 0.157,Y -520.283,Z 1164.314,A 0.000,B 0.000,C 90.000,E1 272.465} C_DIS
LIN {X -0.094,Y -519.671,Z 1164.306,A 0.000,B 0.000,C 90.000,E1 271.031} C_DIS
LIN {X 0.099,Y -518.929,Z 1164.296,A 0.000,B 0.000,C 90.000,E1 269.255} C_DIS
LIN {X -0.176,Y -518.286,Z 1164.288,A 0.000,B 0.000,C 90.000,E1 267.822} C_DIS
LIN {X 0.057,Y -517.457,Z 1164.280,A 0.000,B 0.000,C 90.000,E1 266.331} C_DIS
LIN {X -0.140,Y -516.657,Z 1164.273,A 0.000,B 0.000,C 90.000,E1 265.179} C_DIS
LIN {X 0.197,Y -515.975,Z 1164.268,A 0.000,B 0.000,C 90.000,E1 264.261} C_DIS
LIN {X 0.063,Y -515.152,Z 1164.263,A 0.000,B 0.000,C 90.000,E1 263.394} C_DIS
LIN {X -0.221,Y -513.480,Z 1164.254,A 0.000,B 0.000,C 90.000,E1 261.659} C_DIS
LIN {X -0.149,Y -510.897,Z 1164.239,A 0.000,B 0.000,C 90.000,E1 258.993} C_DIS
LIN {X 0.278,Y -509.547,Z 1164.231,A 0.000,B 0.000,C 90.000,E1 257.465} C_DIS
LIN {X 0.189,Y -508.349,Z 1164.222,A 0.000,B 0.000,C 90.000,E1 255.992} C_DIS
LIN {X 0.073,Y -507.089,Z 1164.214,A 0.000,B 0.000,C 90.000,E1 254.519} C_DIS
LIN {X 0.121,Y -506.027,Z 1164.208,A 0.000,B 0.000,C 90.000,E1 253.323} C_DIS
LIN {X 0.154,Y -504.894,Z 1164.201,A 0.000,B 0.000,C 90.000,E1 252.127} C_DIS
LIN {X -0.233,Y -503.581,Z 1164.193,A 0.000,B 0.000,C 90.000,E1 250.678} C_DIS
LIN {X -0.006,Y -502.128,Z 1164.184,A 0.000,B 0.000,C 90.000,E1 249.156} C_DIS
LIN {X -0.092,Y -500.735,Z 1164.176,A 0.000,B 0.000,C 90.000,E1 247.667} C_DIS
LIN {X 0.122,Y -499.810,Z 1164.171,A 0.000,B 0.000,C 90.000,E1 246.741} C_DIS
LIN {X -0.143,Y -497.226,Z 1164.159,A 0.000,B 0.000,C 90.000,E1 244.665} C_DIS
LIN {X 0.095,Y -495.226,Z 1164.151,A 0.000,B 0.000,C 90.000,E1 243.127} C_DIS
LIN {X -0.143,Y -493.191,Z 1164.142,A 0.000,B 0.000,C 90.000,E1 241.641} C_DIS
LIN {X 0.077,Y -490.136,Z 1164.131,A 0.000,B 0.000,C 90.000,E1 239.488} C_DIS
LIN {X 0.045,Y -487.461,Z 1164.120,A 0.000,B 0.000,C 90.000,E1 237.661} C_DIS
LIN {X 0.224,Y -484.696,Z 1164.110,A 0.000,B 0.000,C 90.000,E1 235.801} C_DIS
LIN {X -0.243,Y -481.558,Z 1164.098,A 0.000,B 0.000,C 90.000,E1 233.703} C_DIS
LIN {X 0.062,Y -479.655,Z 1164.091,A 0.000,B 0.000,C 90.000,E1 232.431} C_DIS
LIN {X -0.150,Y -476.902,Z 1164.081,A 0.000,B 0.000,C 90.000,E1 230.598} C_DIS
LIN {X 0.093,Y -474.725,Z 1164.072,A 0.000,B 0.000,C 90.000,E1 229.013} C_DIS
LIN {X -0.152,Y -472.855,Z 1164.065,A 0.000,B 0.000,C 90.000,E1 227.796} C_DIS
LIN {X -0.023,Y -468.306,Z 1164.050,A 0.000,B 0.000,C 90.000,E1 224.960} C_DIS
LIN {X -0.041,Y -464.815,Z 1164.034,A 0.000,B 0.000,C 90.000,E1 222.123} C_DIS
LIN {X -0.150,Y -461.914,Z 1164.011,A 0.000,B 0.000,C 90.000,E1 218.016} C_DIS
LIN {X -0.135,Y -460.671,Z 1163.995,A 0.000,B 0.000,C 90.000,E1 215.152} C_DIS
LIN {X 0.069,Y -460.371,Z 1163.976,A 0.000,B 0.000,C 90.000,E1 211.623} C_DIS
LIN {X -0.150,Y -462.535,Z 1163.953,A 0.000,B 0.000,C 90.000,E1 207.513} C_DIS
LIN {X -0.020,Y -465.441,Z 1163.937,A 0.000,B 0.000,C 90.000,E1 204.643} C_DIS
LIN {X -0.002,Y -471.068,Z 1163.918,A 0.000,B 0.000,C 90.000,E1 201.173} C_DIS
LIN {X -0.046,Y -478.152,Z 1163.900,A 0.000,B 0.000,C 90.000,E1 198.055} C_DIS
LIN {X -0.129,Y -484.212,Z 1163.888,A 0.000,B 0.000,C 90.000,E1 195.898} C_DIS
LIN {X 0.171,Y -491.060,Z 1163.876,A 0.000,B 0.000,C 90.000,E1 193.716} C_DIS
LIN {X 0.093,Y -499.179,Z 1163.863,A 0.000,B 0.000,C 90.000,E1 191.299} C_DIS
LIN {X -0.047,Y -507.614,Z 1163.850,A 0.000,B 0.000,C 90.000,E1 188.916} C_DIS
LIN {X 0.050,Y -514.165,Z 1163.840,A 0.000,B 0.000,C 90.000,E1 187.125} C_DIS
LIN {X -0.204,Y -519.482,Z 1163.832,A 0.000,B 0.000,C 90.000,E1 185.682} C_DIS
LIN {X 0.106,Y -524.791,Z 1163.823,A 0.000,B 0.000,C 90.000,E1 184.188} C_DIS
LIN {X -0.034,Y -531.149,Z 1163.814,A 0.000,B 0.000,C 90.000,E1 182.465} C_DIS
LIN {X -0.067,Y -535.327,Z 1163.807,A 0.000,B 0.000,C 90.000,E1 181.318} C_DIS
LIN {X -0.038,Y -540.570,Z 1163.799,A 0.000,B 0.000,C 90.000,E1 179.885} C_DIS
LIN {X 0.139,Y -546.880,Z 1163.790,A 0.000,B 0.000,C 90.000,E1 178.165} C_DIS
LIN {X -0.232,Y -551.053,Z 1163.784,A 0.000,B 0.000,C 90.000,E1 177.078} C_DIS
LIN {X 0.196,Y -557.247,Z 1163.774,A 0.000,B 0.000,C 90.000,E1 175.355} C_DIS
LIN {X 0.034,Y -561.404,Z 1163.768,A 0.000,B 0.000,C 90.000,E1 174.261} C_DIS
LIN {X 0.180,Y -567.582,Z 1163.759,A 0.000,B 0.000,C 90.000,E1 172.591} C_DIS
LIN {X 0.237,Y -571.699,Z 1163.753,A 0.000,B 0.000,C 90.000,E1 171.489} C_DIS
LIN {X -0.008,Y -576.744,Z 1163.745,A 0.000,B 0.000,C 90.000,E1 170.151} C_DIS
LIN {X 0.063,Y -582.713,Z 1163.736,A 0.000,B 0.000,C 90.000,E1 168.522} C_DIS
LIN {X -0.127,Y -586.605,Z 1163.730,A 0.000,B 0.000,C 90.000,E1 167.465} C_DIS
LIN {X -0.006,Y -591.311,Z 1163.723,A 0.000,B 0.000,C 90.000,E1 166.117} C_DIS
LIN {X -0.238,Y -595.872,Z 1163.716,A 0.000,B 0.000,C 90.000,E1 164.810} C_DIS
LIN {X -0.105,Y -599.469,Z 1163.710,A 0.000,B 0.000,C 90.000,E1 163.740} C_DIS
LIN {X 0.075,Y -602.903,Z 1163.704,A 0.000,B 0.000,C 90.000,E1 162.670} C_DIS
LIN {X -0.093,Y -606.247,Z 1163.698,A 0.000,B 0.000,C 90.000,E1 161.638} C_DIS
LIN {X 0.096,Y -610.196,Z 1163.691,A 0.000,B 0.000,C 90.000,E1 160.315} C_DIS
LIN {X -0.022,Y -614.050,Z 1163.683,A 0.000,B 0.000,C 90.000,E1 159.028} C_DIS
LIN {X 0.214,Y -616.259,Z 1163.679,A 0.000,B 0.000,C 90.000,E1 158.230} C_DIS
LIN {X -0.138,Y -619.807,Z 1163.672,A 0.000,B 0.000,C 90.000,E1 156.975} C_DIS
LIN {X 0.150,Y -624.009,Z 1163.663,A 0.000,B 0.000,C 90.000,E1 155.409} C_DIS
LIN {X -0.068,Y -627.350,Z 1163.656,A 0.000,B 0.000,C 90.000,E1 154.152} C_DIS
LIN {X 0.038,Y -630.596,Z 1163.649,A 0.000,B 0.000,C 90.000,E1 152.871} C_DIS
LIN {X 0.158,Y -633.134,Z 1163.644,A 0.000,B 0.000,C 90.000,E1 151.847} C_DIS
LIN {X 0.100,Y -636.099,Z 1163.637,A 0.000,B 0.000,C 90.000,E1 150.589} C_DIS
LIN {X 0.098,Y -638.973,Z 1163.630,A 0.000,B 0.000,C 90.000,E1 149.331} C_DIS
LIN {X 0.084,Y -641.092,Z 1163.624,A 0.000,B 0.000,C 90.000,E1 148.329} C_DIS
LIN {X -0.044,Y -643.531,Z 1163.617,A 0.000,B 0.000,C 90.000,E1 147.089} C_DIS
LIN {X 0.410,Y -645.877,Z 1163.610,A 0.000,B 0.000,C 90.000,E1 145.801} C_DIS
LIN {X -0.121,Y -648.482,Z 1163.602,A 0.000,B 0.000,C 90.000,E1 144.356} C_DIS
LIN {X 0.185,Y -650.213,Z 1163.596,A 0.000,B 0.000,C 90.000,E1 143.336} C_DIS
LIN {X 0.056,Y -652.276,Z 1163.590,A 0.000,B 0.000,C 90.000,E1 142.110} C_DIS
LIN {X -0.158,Y -656.286,Z 1163.577,A 0.000,B 0.000,C 90.000,E1 139.908} C_DIS
LIN {X 0.124,Y -660.300,Z 1163.566,A 0.000,B 0.000,C 90.000,E1 137.919} C_DIS
LIN {X 0.034,Y -663.850,Z 1163.557,A 0.000,B 0.000,C 90.000,E1 136.215} C_DIS
LIN {X 0.015,Y -669.548,Z 1163.542,A 0.000,B 0.000,C 90.000,E1 133.542} C_DIS
LIN {X 0.136,Y -673.553,Z 1163.533,A 0.000,B 0.000,C 90.000,E1 131.838} C_DIS
LIN {X -0.050,Y -678.735,Z 1163.521,A 0.000,B 0.000,C 90.000,E1 129.688} C_DIS
LIN {X 0.281,Y -681.737,Z 1163.514,A 0.000,B 0.000,C 90.000,E1 128.463} C_DIS
LIN {X 0.068,Y -683.542,Z 1163.510,A 0.000,B 0.000,C 90.000,E1 127.764} C_DIS
LIN {X -0.022,Y -687.118,Z 1163.502,A 0.000,B 0.000,C 90.000,E1 126.343} C_DIS
LIN {X 0.041,Y -690.066,Z 1163.495,A 0.000,B 0.000,C 90.000,E1 125.152} C_DIS
LIN {X -0.236,Y -692.915,Z 1163.489,A 0.000,B 0.000,C 90.000,E1 123.992} C_DIS
LIN {X -0.108,Y -695.083,Z 1163.484,A 0.000,B 0.000,C 90.000,E1 123.038} C_DIS
LIN {X 0.049,Y -697.169,Z 1163.478,A 0.000,B 0.000,C 90.000,E1 122.084} C_DIS
LIN {X -0.113,Y -699.489,Z 1163.472,A 0.000,B 0.000,C 90.000,E1 120.924} C_DIS
LIN {X 0.001,Y -701.604,Z 1163.465,A 0.000,B 0.000,C 90.000,E1 119.745} C_DIS
LIN {X -0.180,Y -704.077,Z 1163.458,A 0.000,B 0.000,C 90.000,E1 118.359} C_DIS
LIN {X 0.052,Y -705.167,Z 1163.454,A 0.000,B 0.000,C 90.000,E1 117.641} C_DIS
LIN {X -0.029,Y -705.974,Z 1163.450,A 0.000,B 0.000,C 90.000,E1 116.950} C_DIS
LIN {X -0.121,Y -706.518,Z 1163.445,A 0.000,B 0.000,C 90.000,E1 116.027} C_DIS
LIN {X -0.184,Y -706.701,Z 1163.441,A 0.000,B 0.000,C 90.000,E1 115.335} C_DIS
LIN {X 0.109,Y -706.729,Z 1163.439,A 0.000,B 0.000,C 90.000,E1 115.079} C_DIS
LIN {X -0.243,Y -706.450,Z 1163.437,A 0.000,B 0.000,C 90.000,E1 114.643} C_DIS
LIN {X 0.051,Y -705.693,Z 1163.434,A 0.000,B 0.000,C 90.000,E1 114.155} C_DIS
LIN {X -0.303,Y -705.238,Z 1163.433,A 0.000,B 0.000,C 90.000,E1 113.951} C_DIS
LIN {X 0.129,Y -702.675,Z 1163.430,A 0.000,B 0.000,C 90.000,E1 113.334} C_DIS
LIN {X 0.270,Y -701.956,Z 1163.429,A 0.000,B 0.000,C 90.000,E1 113.206} C_DIS
LIN {X -0.106,Y -697.502,Z 1163.427,A 0.000,B 0.000,C 90.000,E1 112.770} C_DIS
LIN {X 0.023,Y -696.173,Z 1163.426,A 0.000,B 0.000,C 90.000,E1 112.642} C_DIS
LIN {X 0.152,Y -694.035,Z 1163.425,A 0.000,B 0.000,C 90.000,E1 112.514} C_DIS
LIN {X -0.042,Y -685.433,Z 1163.424,A 0.000,B 0.000,C 90.000,E1 112.259} C_DIS
LIN {X 0.342,Y -684.093,Z 1163.424,A 0.000,B 0.000,C 90.000,E1 112.206} C_DIS
LIN {X -0.220,Y -676.680,Z 1163.423,A 0.000,B 0.000,C 90.000,E1 112.206} C_DIS
LIN {X -0.246,Y -604.396,Z 1163.423,A 0.000,B 0.000,C 90.000,E1 112.206} C_DIS
LIN {X -0.200,Y -600.848,Z 1163.422,A 0.000,B 0.000,C 90.000,E1 111.972} C_DIS
LIN {X 0.026,Y -595.412,Z 1163.420,A 0.000,B 0.000,C 90.000,E1 111.535} C_DIS
LIN {X -0.116,Y -578.287,Z 1163.411,A 0.000,B 0.000,C 90.000,E1 110.066} C_DIS
LIN {X -0.077,Y -573.972,Z 1163.409,A 0.000,B 0.000,C 90.000,E1 109.704} C_DIS
LIN {X -0.259,Y -568.033,Z 1163.407,A 0.000,B 0.000,C 90.000,E1 109.268} C_DIS
LIN {X -0.165,Y -560.164,Z 1163.404,A 0.000,B 0.000,C 90.000,E1 108.725} C_DIS
LIN {X -0.148,Y -555.520,Z 1163.402,A 0.000,B 0.000,C 90.000,E1 108.417} C_DIS
LIN {X -0.171,Y -551.711,Z 1163.401,A 0.000,B 0.000,C 90.000,E1 108.109} C_DIS
LIN {X 0.026,Y -550.382,Z 1163.399,A 0.000,B 0.000,C 90.000,E1 107.873} C_DIS
LIN {X -0.014,Y -550.365,Z 1163.399,A 0.000,B 0.000,C 90.000,E1 107.873} C_DIS
LIN {X -0.119,Y -550.020,Z 1163.398,A 0.000,B 0.000,C 90.000,E1 107.583} C_DIS
LIN {X -0.230,Y -550.049,Z 1163.396,A 0.000,B 0.000,C 90.000,E1 107.275} C_DIS
LIN {X -0.116,Y -551.542,Z 1163.385,A 0.000,B 0.000,C 90.000,E1 105.300} C_DIS
LIN {X 0.165,Y -552.947,Z 1163.376,A 0.000,B 0.000,C 90.000,E1 103.592} C_DIS
LIN {X 0.078,Y -555.006,Z 1163.363,A 0.000,B 0.000,C 90.000,E1 101.366} C_DIS
LIN {X 0.055,Y -556.154,Z 1163.357,A 0.000,B 0.000,C 90.000,E1 100.254} C_DIS
LIN {X 0.217,Y -557.722,Z 1163.348,A 0.000,B 0.000,C 90.000,E1 98.568} C_DIS
LIN {X 0.191,Y -558.956,Z 1163.340,A 0.000,B 0.000,C 90.000,E1 97.182} C_DIS
LIN {X -0.159,Y -560.397,Z 1163.329,A 0.000,B 0.000,C 90.000,E1 95.277} C_DIS
LIN {X -0.110,Y -561.554,Z 1163.320,A 0.000,B 0.000,C 90.000,E1 93.612} C_DIS
LIN {X -0.059,Y -562.801,Z 1163.311,A 0.000,B 0.000,C 90.000,E1 91.949} C_DIS
LIN {X 0.018,Y -564.072,Z 1163.302,A 0.000,B 0.000,C 90.000,E1 90.286} C_DIS
LIN {X -0.113,Y -564.854,Z 1163.296,A 0.000,B 0.000,C 90.000,E1 89.198} C_DIS
LIN {X -0.108,Y -565.720,Z 1163.288,A 0.000,B 0.000,C 90.000,E1 87.822} C_DIS
LIN {X 0.026,Y -566.721,Z 1163.279,A 0.000,B 0.000,C 90.000,E1 86.159} C_DIS
LIN {X 0.259,Y -567.712,Z 1163.270,A 0.000,B 0.000,C 90.000,E1 84.489} C_DIS
LIN {X -0.043,Y -568.820,Z 1163.260,A 0.000,B 0.000,C 90.000,E1 82.875} C_DIS
LIN {X 0.128,Y -569.609,Z 1163.253,A 0.000,B 0.000,C 90.000,E1 81.489} C_DIS
LIN {X 0.021,Y -570.391,Z 1163.244,A 0.000,B 0.000,C 90.000,E1 79.859} C_DIS
LIN {X -0.070,Y -571.235,Z 1163.235,A 0.000,B 0.000,C 90.000,E1 78.229} C_DIS
LIN {X -0.075,Y -572.275,Z 1163.223,A 0.000,B 0.000,C 90.000,E1 76.047} C_DIS
LIN {X 0.116,Y -573.062,Z 1163.213,A 0.000,B 0.000,C 90.000,E1 74.393} C_DIS
LIN {X -0.083,Y -574.397,Z 1163.201,A 0.000,B 0.000,C 90.000,E1 72.236} C_DIS
LIN {X -0.065,Y -576.301,Z 1163.186,A 0.000,B 0.000,C 90.000,E1 69.518} C_DIS
LIN {X 0.005,Y -577.929,Z 1163.176,A 0.000,B 0.000,C 90.000,E1 67.614} C_DIS
LIN {X 0.181,Y -579.555,Z 1163.167,A 0.000,B 0.000,C 90.000,E1 65.973} C_DIS
LIN {X 0.152,Y -581.014,Z 1163.158,A 0.000,B 0.000,C 90.000,E1 64.357} C_DIS
LIN {X -0.007,Y -582.796,Z 1163.147,A 0.000,B 0.000,C 90.000,E1 62.487} C_DIS
LIN {X 0.004,Y -584.259,Z 1163.138,A 0.000,B 0.000,C 90.000,E1 60.873} C_DIS
LIN {X -0.058,Y -585.371,Z 1163.131,A 0.000,B 0.000,C 90.000,E1 59.537} C_DIS
LIN {X 0.034,Y -586.161,Z 1163.125,A 0.000,B 0.000,C 90.000,E1 58.456} C_DIS
LIN {X 0.010,Y -587.129,Z 1163.117,A 0.000,B 0.000,C 90.000,E1 57.120} C_DIS
LIN {X -0.370,Y -587.908,Z 1163.111,A 0.000,B 0.000,C 90.000,E1 56.087} C_DIS
LIN {X -0.345,Y -588.866,Z 1163.103,A 0.000,B 0.000,C 90.000,E1 54.482} C_DIS
LIN {X 0.250,Y -590.018,Z 1163.092,A 0.000,B 0.000,C 90.000,E1 52.557} C_DIS
LIN {X -0.061,Y -591.052,Z 1163.082,A 0.000,B 0.000,C 90.000,E1 50.723} C_DIS
LIN {X -0.141,Y -591.531,Z 1163.076,A 0.000,B 0.000,C 90.000,E1 49.666} C_DIS
LIN {X -0.250,Y -591.933,Z 1163.067,A 0.000,B 0.000,C 90.000,E1 48.081} C_DIS
LIN {X 0.076,Y -592.064,Z 1163.061,A 0.000,B 0.000,C 90.000,E1 46.986} C_DIS
LIN {X 0.402,Y -592.032,Z 1163.055,A 0.000,B 0.000,C 90.000,E1 45.891} C_DIS
LIN {X 0.301,Y -591.853,Z 1163.049,A 0.000,B 0.000,C 90.000,E1 44.838} C_DIS
LIN {X 0.196,Y -591.448,Z 1163.043,A 0.000,B 0.000,C 90.000,E1 43.785} C_DIS
LIN {X 0.270,Y -590.764,Z 1163.036,A 0.000,B 0.000,C 90.000,E1 42.447} C_DIS
LIN {X -0.017,Y -590.197,Z 1163.032,A 0.000,B 0.000,C 90.000,E1 41.676} C_DIS
LIN {X -0.168,Y -588.581,Z 1163.023,A 0.000,B 0.000,C 90.000,E1 40.092} C_DIS
LIN {X 0.166,Y -587.320,Z 1163.017,A 0.000,B 0.000,C 90.000,E1 38.991} C_DIS
LIN {X 0.022,Y -585.920,Z 1163.011,A 0.000,B 0.000,C 90.000,E1 37.935} C_DIS
LIN {X -0.043,Y -584.225,Z 1163.005,A 0.000,B 0.000,C 90.000,E1 36.870} C_DIS
LIN {X -0.127,Y -582.189,Z 1162.999,A 0.000,B 0.000,C 90.000,E1 35.804} C_DIS
LIN {X 0.064,Y -580.313,Z 1162.994,A 0.000,B 0.000,C 90.000,E1 34.978} C_DIS
LIN {X -0.240,Y -578.244,Z 1162.990,A 0.000,B 0.000,C 90.000,E1 34.199} C_DIS
LIN {X -0.088,Y -575.787,Z 1162.985,A 0.000,B 0.000,C 90.000,E1 33.372} C_DIS
LIN {X -0.106,Y -574.050,Z 1162.982,A 0.000,B 0.000,C 90.000,E1 32.832} C_DIS
LIN {X -0.002,Y -571.016,Z 1162.978,A 0.000,B 0.000,C 90.000,E1 32.005} C_DIS
LIN {X -0.054,Y -568.818,Z 1162.975,A 0.000,B 0.000,C 90.000,E1 31.465} C_DIS
LIN {X -0.305,Y -565.082,Z 1162.970,A 0.000,B 0.000,C 90.000,E1 30.669} C_DIS
LIN {X 0.182,Y -563.089,Z 1162.968,A 0.000,B 0.000,C 90.000,E1 30.207} C_DIS
LIN {X -0.235,Y -558.035,Z 1162.963,A 0.000,B 0.000,C 90.000,E1 29.283} C_DIS
LIN {X -0.113,Y -553.261,Z 1162.958,A 0.000,B 0.000,C 90.000,E1 28.437} C_DIS
LIN {X 0.070,Y -548.999,Z 1162.954,A 0.000,B 0.000,C 90.000,E1 27.719} C_DIS
LIN {X 0.212,Y -544.406,Z 1162.950,A 0.000,B 0.000,C 90.000,E1 27.001} C_DIS
LIN {X 0.064,Y -539.234,Z 1162.946,A 0.000,B 0.000,C 90.000,E1 26.309} C_DIS
LIN {X 0.111,Y -533.706,Z 1162.942,A 0.000,B 0.000,C 90.000,E1 25.591} C_DIS
LIN {X -0.126,Y -527.897,Z 1162.938,A 0.000,B 0.000,C 90.000,E1 24.899} C_DIS
LIN {X 0.071,Y -521.595,Z 1162.934,A 0.000,B 0.000,C 90.000,E1 24.155} C_DIS
LIN {X -0.014,Y -516.417,Z 1162.931,A 0.000,B 0.000,C 90.000,E1 23.590} C_DIS
LIN {X -0.041,Y -509.850,Z 1162.927,A 0.000,B 0.000,C 90.000,E1 22.898} C_DIS
LIN {X -0.001,Y -501.821,Z 1162.923,A 0.000,B 0.000,C 90.000,E1 22.078} C_DIS
LIN {X -0.091,Y -492.024,Z 1162.917,A 0.000,B 0.000,C 90.000,E1 21.153} C_DIS
LIN {X 0.131,Y -480.328,Z 1162.912,A 0.000,B 0.000,C 90.000,E1 20.066} C_DIS
LIN {X -0.113,Y -468.525,Z 1162.906,A 0.000,B 0.000,C 90.000,E1 19.033} C_DIS
LIN {X -0.213,Y -452.152,Z 1162.898,A 0.000,B 0.000,C 90.000,E1 17.583} C_DIS
LIN {X -0.150,Y -431.809,Z 1162.887,A 0.000,B 0.000,C 90.000,E1 15.607} C_DIS
LIN {X 0.086,Y -416.326,Z 1162.877,A 0.000,B 0.000,C 90.000,E1 13.883} C_DIS
LIN {X -0.138,Y -406.950,Z 1162.871,A 0.000,B 0.000,C 90.000,E1 12.771} C_DIS
LIN {X -0.091,Y -398.459,Z 1162.864,A 0.000,B 0.000,C 90.000,E1 11.591} C_DIS
LIN {X -0.013,Y -395.781,Z 1162.862,A 0.000,B 0.000,C 90.000,E1 11.130} C_DIS
LIN {X 0.016,Y -394.887,Z 1162.861,A 0.000,B 0.000,C 90.000,E1 10.950} C_DIS
LIN {X -0.045,Y -393.123,Z 1162.859,A 0.000,B 0.000,C 90.000,E1 10.546} C_DIS
LIN {X -0.083,Y -393.118,Z 1162.859,A 0.000,B 0.000,C 90.000,E1 10.546} C_DIS
LIN {X -0.114,Y -392.593,Z 1162.856,A 0.000,B 0.000,C 90.000,E1 10.141} C_DIS
LIN {X -0.152,Y -392.598,Z 1162.856,A 0.000,B 0.000,C 90.000,E1 10.141} C_DIS
LIN {X 0.137,Y -393.528,Z 1162.853,A 0.000,B 0.000,C 90.000,E1 9.500} C_DIS
LIN {X 0.071,Y -396.026,Z 1162.848,A 0.000,B 0.000,C 90.000,E1 8.624} C_DIS
LIN {X -0.050,Y -398.392,Z 1162.844,A 0.000,B 0.000,C 90.000,E1 7.936} C_DIS
LIN {X -0.123,Y -401.837,Z 1162.839,A 0.000,B 0.000,C 90.000,E1 7.068} C_DIS
LIN {X -0.133,Y -403.822,Z 1162.837,A 0.000,B 0.000,C 90.000,E1 6.720} C_DIS
LIN {X -0.163,Y -406.974,Z 1162.834,A 0.000,B 0.000,C 90.000,E1 6.201} C_DIS
LIN {X -0.004,Y -411.092,Z 1162.832,A 0.000,B 0.000,C 90.000,E1 5.739} C_DIS
LIN {X -0.096,Y -416.468,Z 1162.830,A 0.000,B 0.000,C 90.000,E1 5.334} C_DIS
LIN {X -0.148,Y -432.684,Z 1162.823,A 0.000,B 0.000,C 90.000,E1 4.131} C_DIS
LIN {X 0.197,Y -447.146,Z 1162.817,A 0.000,B 0.000,C 90.000,E1 3.037} C_DIS
LIN {X -0.027,Y -464.998,Z 1162.810,A 0.000,B 0.000,C 90.000,E1 1.835} C_DIS
LIN {X 0.158,Y -476.126,Z 1162.806,A 0.000,B 0.000,C 90.000,E1 1.031} C_DIS
LIN {X 0.171,Y -485.387,Z 1162.802,A 0.000,B 0.000,C 90.000,E1 0.344} C_DIS
LIN {X 0.000,Y -490.212,Z 1162.800,A 0.000,B 0.000,C 90.000,E1 360.000} C_DIS
LIN {X -0.065,Y -497.223,Z 1162.797,A 0.000,B 0.000,C 90.000,E1 359.427} C_DIS
LIN {X 0.055,Y -504.074,Z 1162.793,A 0.000,B 0.000,C 90.000,E1 358.797} C_DIS
LIN {X 0.240,Y -510.857,Z 1162.790,A 0.000,B 0.000,C 90.000,E1 358.108} C_DIS
LIN {X -0.132,Y -516.126,Z 1162.787,A 0.000,B 0.000,C 90.000,E1 357.593} C_DIS
LIN {X -0.251,Y -522.251,Z 1162.783,A 0.000,B 0.000,C 90.000,E1 356.906} C_DIS
LIN {X -0.058,Y -528.079,Z 1162.779,A 0.000,B 0.000,C 90.000,E1 356.159} C_DIS
LIN {X -0.083,Y -532.353,Z 1162.776,A 0.000,B 0.000,C 90.000,E1 355.584} C_DIS
LIN {X 0.188,Y -537.099,Z 1162.771,A 0.000,B 0.000,C 90.000,E1 354.837} C_DIS
LIN {X -0.033,Y -541.393,Z 1162.767,A 0.000,B 0.000,C 90.000,E1 354.147} C_DIS
LIN {X -0.160,Y -545.262,Z 1162.764,A 0.000,B 0.000,C 90.000,E1 353.451} C_DIS
LIN {X -0.055,Y -548.114,Z 1162.760,A 0.000,B 0.000,C 90.000,E1 352.875} C_DIS
LIN {X 0.175,Y -552.009,Z 1162.756,A 0.000,B 0.000,C 90.000,E1 352.008} C_DIS
LIN {X -0.222,Y -554.340,Z 1162.753,A 0.000,B 0.000,C 90.000,E1 351.489} C_DIS
LIN {X 0.024,Y -556.471,Z 1162.750,A 0.000,B 0.000,C 90.000,E1 350.905} C_DIS
LIN {X -0.215,Y -559.380,Z 1162.745,A 0.000,B 0.000,C 90.000,E1 350.095} C_DIS
LIN {X 0.225,Y -562.060,Z 1162.740,A 0.000,B 0.000,C 90.000,E1 349.218} C_DIS
LIN {X 0.034,Y -564.473,Z 1162.736,A 0.000,B 0.000,C 90.000,E1 348.409} C_DIS
LIN {X 0.145,Y -567.541,Z 1162.730,A 0.000,B 0.000,C 90.000,E1 347.297} C_DIS
LIN {X 0.059,Y -570.990,Z 1162.722,A 0.000,B 0.000,C 90.000,E1 345.936} C_DIS
LIN {X -0.153,Y -573.644,Z 1162.716,A 0.000,B 0.000,C 90.000,E1 344.866} C_DIS
LIN {X -0.130,Y -576.687,Z 1162.708,A 0.000,B 0.000,C 90.000,E1 343.504} C_DIS
LIN {X -0.067,Y -580.238,Z 1162.699,A 0.000,B 0.000,C 90.000,E1 341.873} C_DIS
LIN {X 0.176,Y -581.824,Z 1162.695,A 0.000,B 0.000,C 90.000,E1 341.040} C_DIS
LIN {X -0.272,Y -583.810,Z 1162.689,A 0.000,B 0.000,C 90.000,E1 340.007} C_DIS
LIN {X -0.075,Y -585.953,Z 1162.681,A 0.000,B 0.000,C 90.000,E1 338.646} C_DIS
LIN {X -0.004,Y -586.680,Z 1162.678,A 0.000,B 0.000,C 90.000,E1 338.103} C_DIS
LIN {X -0.178,Y -587.849,Z 1162.672,A 0.000,B 0.000,C 90.000,E1 337.050} C_DIS
LIN {X 0.011,Y -588.425,Z 1162.668,A 0.000,B 0.000,C 90.000,E1 336.230} C_DIS
LIN {X 0.322,Y -588.684,Z 1162.665,A 0.000,B 0.000,C 90.000,E1 335.665} C_DIS
LIN {X -0.258,Y -588.789,Z 1162.661,A 0.000,B 0.000,C 90.000,E1 334.921} C_DIS
LIN {X -0.060,Y -588.624,Z 1162.656,A 0.000,B 0.000,C 90.000,E1 334.101} C_DIS
LIN {X -0.020,Y -588.376,Z 1162.653,A 0.000,B 0.000,C 90.000,E1 333.563} C_DIS
LIN {X 0.173,Y -587.553,Z 1162.649,A 0.000,B 0.000,C 90.000,E1 332.743} C_DIS
LIN {X -0.053,Y -586.895,Z 1162.646,A 0.000,B 0.000,C 90.000,E1 332.231} C_DIS
LIN {X -0.009,Y -585.963,Z 1162.643,A 0.000,B 0.000,C 90.000,E1 331.691} C_DIS
LIN {X 0.142,Y -584.316,Z 1162.638,A 0.000,B 0.000,C 90.000,E1 330.873} C_DIS
LIN {X 0.043,Y -582.292,Z 1162.634,A 0.000,B 0.000,C 90.000,E1 330.078} C_DIS
LIN {X -0.074,Y -579.731,Z 1162.629,A 0.000,B 0.000,C 90.000,E1 329.282} C_DIS
LIN {X 0.082,Y -576.624,Z 1162.625,A 0.000,B 0.000,C 90.000,E1 328.456} C_DIS
LIN {X -0.098,Y -572.447,Z 1162.620,A 0.000,B 0.000,C 90.000,E1 327.661} C_DIS
LIN {X -0.143,Y -569.398,Z 1162.617,A 0.000,B 0.000,C 90.000,E1 327.120} C_DIS
LIN {X 0.000,Y -564.852,Z 1162.614,A 0.000,B 0.000,C 90.000,E1 326.421} C_DIS
LIN {X 0.110,Y -560.003,Z 1162.610,A 0.000,B 0.000,C 90.000,E1 325.722} C_DIS
LIN {X 0.090,Y -556.850,Z 1162.607,A 0.000,B 0.000,C 90.000,E1 325.308} C_DIS
LIN {X 0.010,Y -548.814,Z 1162.602,A 0.000,B 0.000,C 90.000,E1 324.356} C_DIS
LIN {X 0.289,Y -542.551,Z 1162.598,A 0.000,B 0.000,C 90.000,E1 323.623} C_DIS
LIN {X -0.091,Y -533.512,Z 1162.593,A 0.000,B 0.000,C 90.000,E1 322.683} C_DIS
LIN {X 0.049,Y -528.801,Z 1162.590,A 0.000,B 0.000,C 90.000,E1 322.145} C_DIS
LIN {X 0.034,Y -526.453,Z 1162.588,A 0.000,B 0.000,C 90.000,E1 321.859} C_DIS
LIN {X -0.012,Y -523.724,Z 1162.586,A 0.000,B 0.000,C 90.000,E1 321.492} C_DIS
LIN {X 0.093,Y -521.345,Z 1162.584,A 0.000,B 0.000,C 90.000,E1 321.045} C_DIS
LIN {X -0.219,Y -519.698,Z 1162.581,A 0.000,B 0.000,C 90.000,E1 320.642} C_DIS
LIN {X -0.080,Y -519.236,Z 1162.580,A 0.000,B 0.000,C 90.000,E1 320.481} C_DIS
LIN {X 0.261,Y -518.218,Z 1162.577,A 0.000,B 0.000,C 90.000,E1 319.828} C_DIS
LIN {X -0.189,Y -518.085,Z 1162.575,A 0.000,B 0.000,C 90.000,E1 319.542} C_DIS
LIN {X 0.225,Y -518.270,Z 1162.569,A 0.000,B 0.000,C 90.000,E1 318.324} C_DIS
LIN {X 0.092,Y -519.111,Z 1162.559,A 0.000,B 0.000,C 90.000,E1 316.581} C_DIS
LIN {X -0.018,Y -519.987,Z 1162.549,A 0.000,B 0.000,C 90.000,E1 314.838} C_DIS
LIN {X -0.110,Y -520.865,Z 1162.539,A 0.000,B 0.000,C 90.000,E1 313.095} C_DIS
LIN {X -0.248,Y -522.029,Z 1162.528,A 0.000,B 0.000,C 90.000,E1 311.067} C_DIS
LIN {X 0.134,Y -523.015,Z 1162.518,A 0.000,B 0.000,C 90.000,E1 309.277} C_DIS
LIN {X 0.251,Y -523.867,Z 1162.510,A 0.000,B 0.000,C 90.000,E1 307.810} C_DIS
LIN {X 0.062,Y -524.808,Z 1162.502,A 0.000,B 0.000,C 90.000,E1 306.377} C_DIS
LIN {X 0.245,Y -525.934,Z 1162.491,A 0.000,B 0.000,C 90.000,E1 304.326} C_DIS
LIN {X 0.268,Y -527.404,Z 1162.478,A 0.000,B 0.000,C 90.000,E1 302.005} C_DIS
LIN {X -0.328,Y -528.450,Z 1162.468,A 0.000,B 0.000,C 90.000,E1 300.335} C_DIS
LIN {X 0.201,Y -528.920,Z 1162.464,A 0.000,B 0.000,C 90.000,E1 299.411} C_DIS
LIN {X 0.134,Y -529.527,Z 1162.456,A 0.000,B 0.000,C 90.000,E1 297.975} C_DIS
LIN {X -0.046,Y -529.785,Z 1162.451,A 0.000,B 0.000,C 90.000,E1 297.129} C_DIS
LIN {X 0.131,Y -530.040,Z 1162.443,A 0.000,B 0.000,C 90.000,E1 295.668} C_DIS
LIN {X -0.170,Y -530.073,Z 1162.435,A 0.000,B 0.000,C 90.000,E1 294.259} C_DIS
LIN {X 0.159,Y -530.023,Z 1162.423,A 0.000,B 0.000,C 90.000,E1 292.206} C_DIS
LIN {X -0.087,Y -529.928,Z 1162.416,A 0.000,B 0.000,C 90.000,E1 290.791} C_DIS
LIN {X 0.166,Y -529.452,Z 1162.406,A 0.000,B 0.000,C 90.000,E1 289.033} C_DIS
LIN {X 0.217,Y -529.082,Z 1162.400,A 0.000,B 0.000,C 90.000,E1 287.873} C_DIS
LIN {X 0.113,Y -528.506,Z 1162.391,A 0.000,B 0.000,C 90.000,E1 286.441} C_DIS
LIN {X -0.022,Y -528.047,Z 1162.385,A 0.000,B 0.000,C 90.000,E1 285.300} C_DIS
LIN {X -0.263,Y -527.092,Z 1162.375,A 0.000,B 0.000,C 90.000,E1 283.592} C_DIS
LIN {X -0.052,Y -526.404,Z 1162.369,A 0.000,B 0.000,C 90.000,E1 282.411} C_DIS
LIN {X 0.052,Y -525.485,Z 1162.361,A 0.000,B 0.000,C 90.000,E1 280.950} C_DIS
LIN {X 0.049,Y -524.485,Z 1162.353,A 0.000,B 0.000,C 90.000,E1 279.500} C_DIS
LIN {X 0.041,Y -523.387,Z 1162.343,A 0.000,B 0.000,C 90.000,E1 277.757} C_DIS
LIN {X -0.130,Y -522.328,Z 1162.333,A 0.000,B 0.000,C 90.000,E1 276.030} C_DIS
LIN {X 0.203,Y -521.485,Z 1162.324,A 0.000,B 0.000,C 90.000,E1 274.245} C_DIS
LIN {X -0.048,Y -520.722,Z 1162.314,A 0.000,B 0.000,C 90.000,E1 272.522} C_DIS
LIN {X -0.238,Y -520.255,Z 1162.307,A 0.000,B 0.000,C 90.000,E1 271.375} C_DIS
LIN {X -0.089,Y -519.395,Z 1162.296,A 0.000,B 0.000,C 90.000,E1 269.312} C_DIS
LIN {X 0.165,Y -518.756,Z 1162.288,A 0.000,B 0.000,C 90.000,E1 267.822} C_DIS
LIN {X -0.111,Y -517.937,Z 1162.280,A 0.000,B 0.000,C 90.000,E1 266.388} C_DIS
LIN {X 0.215,Y -517.150,Z 1162.273,A 0.000,B 0.000,C 90.000,E1 265.179} C_DIS
LIN {X -0.059,Y -515.998,Z 1162.265,A 0.000,B 0.000,C 90.000,E1 263.742} C_DIS
LIN {X 0.155,Y -513.953,Z 1162.254,A 0.000,B 0.000,C 90.000,E1 261.659} C_DIS
LIN {X -0.052,Y -512.476,Z 1162.246,A 0.000,B 0.000,C 90.000,E1 260.208} C_DIS
LIN {X 0.141,Y -510.587,Z 1162.234,A 0.000,B 0.000,C 90.000,E1 258.117} C_DIS
LIN {X 0.057,Y -508.544,Z 1162.221,A 0.000,B 0.000,C 90.000,E1 255.755} C_DIS
LIN {X 0.027,Y -507.014,Z 1162.211,A 0.000,B 0.000,C 90.000,E1 253.976} C_DIS
LIN {X 0.098,Y -505.404,Z 1162.201,A 0.000,B 0.000,C 90.000,E1 252.181} C_DIS
LIN {X -0.193,Y -503.744,Z 1162.191,A 0.000,B 0.000,C 90.000,E1 250.423} C_DIS
LIN {X 0.200,Y -501.707,Z 1162.180,A 0.000,B 0.000,C 90.000,E1 248.284} C_DIS
LIN {X 0.039,Y -500.515,Z 1162.173,A 0.000,B 0.000,C 90.000,E1 247.102} C_DIS
LIN {X -0.140,Y -499.077,Z 1162.166,A 0.000,B 0.000,C 90.000,E1 245.921} C_DIS
LIN {X -0.135,Y -497.642,Z 1162.160,A 0.000,B 0.000,C 90.000,E1 244.717} C_DIS
LIN {X -0.107,Y -495.637,Z 1162.151,A 0.000,B 0.000,C 90.000,E1 243.204} C_DIS
LIN {X -0.109,Y -493.585,Z 1162.143,A 0.000,B 0.000,C 90.000,E1 241.691} C_DIS
LIN {X -0.039,Y -490.046,Z 1162.129,A 0.000,B 0.000,C 90.000,E1 239.253} C_DIS
LIN {X 0.114,Y -487.781,Z 1162.121,A 0.000,B 0.000,C 90.000,E1 237.709} C_DIS
LIN {X 0.036,Y -485.024,Z 1162.110,A 0.000,B 0.000,C 90.000,E1 235.881} C_DIS
LIN {X 0.247,Y -481.865,Z 1162.099,A 0.000,B 0.000,C 90.000,E1 233.703} C_DIS
LIN {X 0.175,Y -479.973,Z 1162.092,A 0.000,B 0.000,C 90.000,E1 232.477} C_DIS
LIN {X -0.223,Y -476.664,Z 1162.080,A 0.000,B 0.000,C 90.000,E1 230.356} C_DIS
LIN {X 0.020,Y -474.424,Z 1162.071,A 0.000,B 0.000,C 90.000,E1 228.771} C_DIS
LIN {X -0.228,Y -472.466,Z 1162.064,A 0.000,B 0.000,C 90.000,E1 227.553} C_DIS
LIN {X 0.064,Y -468.902,Z 1162.052,A 0.000,B 0.000,C 90.000,E1 225.324} C_DIS
LIN {X 0.207,Y -464.559,Z 1162.033,A 0.000,B 0.000,C 90.000,E1 221.838} C_DIS
LIN {X -0.050,Y -461.997,Z 1162.013,A 0.000,B 0.000,C 90.000,E1 218.382} C_DIS
LIN {X 0.094,Y -460.966,Z 1162.003,A 0.000,B 0.000,C 90.000,E1 216.457} C_DIS
LIN {X 0.193,Y -459.992,Z 1161.987,A 0.000,B 0.000,C 90.000,E1 213.579} C_DIS
LIN {X -0.116,Y -460.059,Z 1161.974,A 0.000,B 0.000,C 90.000,E1 211.386} C_DIS
LIN {X -0.110,Y -463.319,Z 1161.944,A 0.000,B 0.000,C 90.000,E1 205.976} C_DIS
LIN {X -0.212,Y -466.051,Z 1161.932,A 0.000,B 0.000,C 90.000,E1 203.770} C_DIS
LIN {X -0.167,Y -472.223,Z 1161.913,A 0.000,B 0.000,C 90.000,E1 200.301} C_DIS
LIN {X 0.142,Y -479.097,Z 1161.897,A 0.000,B 0.000,C 90.000,E1 197.457} C_DIS
LIN {X -0.184,Y -488.373,Z 1161.880,A 0.000,B 0.000,C 90.000,E1 194.411} C_DIS
LIN {X -0.060,Y -492.374,Z 1161.873,A 0.000,B 0.000,C 90.000,E1 193.175} C_DIS
LIN {X -0.235,Y -499.599,Z 1161.861,A 0.000,B 0.000,C 90.000,E1 191.074} C_DIS
LIN {X -0.218,Y -507.041,Z 1161.850,A 0.000,B 0.000,C 90.000,E1 188.973} C_DIS
LIN {X -0.138,Y -513.633,Z 1161.840,A 0.000,B 0.000,C 90.000,E1 187.182} C_DIS
LIN {X 0.188,Y -517.935,Z 1161.833,A 0.000,B 0.000,C 90.000,E1 185.967} C_DIS
LIN {X -0.055,Y -523.267,Z 1161.825,A 0.000,B 0.000,C 90.000,E1 184.531} C_DIS
LIN {X -0.205,Y -528.597,Z 1161.817,A 0.000,B 0.000,C 90.000,E1 183.094} C_DIS
LIN {X 0.236,Y -532.856,Z 1161.811,A 0.000,B 0.000,C 90.000,E1 181.892} C_DIS
LIN {X 0.245,Y -539.179,Z 1161.801,A 0.000,B 0.000,C 90.000,E1 180.172} C_DIS
LIN {X -0.196,Y -544.450,Z 1161.793,A 0.000,B 0.000,C 90.000,E1 178.797} C_DIS
LIN {X 0.058,Y -550.816,Z 1161.784,A 0.000,B 0.000,C 90.000,E1 177.078} C_DIS
LIN {X 0.045,Y -558.135,Z 1161.773,A 0.000,B 0.000,C 90.000,E1 175.122} C_DIS
LIN {X -0.158,Y -562.286,Z 1161.767,A 0.000,B 0.000,C 90.000,E1 174.033} C_DIS
LIN {X 0.073,Y -568.502,Z 1161.758,A 0.000,B 0.000,C 90.000,E1 172.356} C_DIS
LIN {X 0.148,Y -572.619,Z 1161.752,A 0.000,B 0.000,C 90.000,E1 171.254} C_DIS
LIN {X 0.284,Y -576.737,Z 1161.745,A 0.000,B 0.000,C 90.000,E1 170.151} C_DIS
LIN {X -0.215,Y -582.772,Z 1161.736,A 0.000,B 0.000,C 90.000,E1 168.578} C_DIS
LIN {X -0.156,Y -587.650,Z 1161.729,A 0.000,B 0.000,C 90.000,E1 167.229} C_DIS
LIN {X -0.016,Y -592.372,Z 1161.722,A 0.000,B 0.000,C 90.000,E1 165.880} C_DIS
LIN {X 0.049,Y -597.828,Z 1161.713,A 0.000,B 0.000,C 90.000,E1 164.283} C_DIS
LIN {X 0.094,Y -602.250,Z 1161.705,A 0.000,B 0.000,C 90.000,E1 162.960} C_DIS
LIN {X 0.224,Y -606.416,Z 1161.698,A 0.000,B 0.000,C 90.000,E1 161.638} C_DIS
LIN {X -0.217,Y -611.155,Z 1161.689,A 0.000,B 0.000,C 90.000,E1 160.115} C_DIS
LIN {X 0.004,Y -615.695,Z 1161.681,A 0.000,B 0.000,C 90.000,E1 158.539} C_DIS
LIN {X 0.195,Y -619.941,Z 1161.672,A 0.000,B 0.000,C 90.000,E1 156.975} C_DIS
LIN {X -0.084,Y -623.438,Z 1161.665,A 0.000,B 0.000,C 90.000,E1 155.717} C_DIS
LIN {X 0.273,Y -627.428,Z 1161.657,A 0.000,B 0.000,C 90.000,E1 154.152} C_DIS
LIN {X -0.180,Y -630.645,Z 1161.650,A 0.000,B 0.000,C 90.000,E1 152.922} C_DIS
LIN {X -0.054,Y -633.183,Z 1161.644,A 0.000,B 0.000,C 90.000,E1 151.897} C_DIS
LIN {X -0.105,Y -636.118,Z 1161.637,A 0.000,B 0.000,C 90.000,E1 150.639} C_DIS
LIN {X -0.102,Y -638.985,Z 1161.630,A 0.000,B 0.000,C 90.000,E1 149.380} C_DIS
LIN {X -0.057,Y -641.543,Z 1161.623,A 0.000,B 0.000,C 90.000,E1 148.122} C_DIS
LIN {X 0.364,Y -643.966,Z 1161.616,A 0.000,B 0.000,C 90.000,E1 146.834} C_DIS
LIN {X -0.135,Y -645.844,Z 1161.610,A 0.000,B 0.000,C 90.000,E1 145.881} C_DIS
LIN {X -0.294,Y -648.440,Z 1161.602,A 0.000,B 0.000,C 90.000,E1 144.402} C_DIS
LIN {X -0.371,Y -650.163,Z 1161.597,A 0.000,B 0.000,C 90.000,E1 143.417} C_DIS
LIN {X -0.058,Y -652.621,Z 1161.588,A 0.000,B 0.000,C 90.000,E1 141.904} C_DIS
LIN {X 0.196,Y -656.199,Z 1161.577,A 0.000,B 0.000,C 90.000,E1 139.908} C_DIS
LIN {X 0.037,Y -660.214,Z 1161.567,A 0.000,B 0.000,C 90.000,E1 137.957} C_DIS
LIN {X 0.388,Y -663.741,Z 1161.557,A 0.000,B 0.000,C 90.000,E1 136.215} C_DIS
LIN {X 0.362,Y -668.894,Z 1161.543,A 0.000,B 0.000,C 90.000,E1 133.785} C_DIS
LIN {X -0.013,Y -673.423,Z 1161.533,A 0.000,B 0.000,C 90.000,E1 131.881} C_DIS
LIN {X -0.131,Y -678.604,Z 1161.521,A 0.000,B 0.000,C 90.000,E1 129.725} C_DIS
LIN {X -0.326,Y -681.640,Z 1161.514,A 0.000,B 0.000,C 90.000,E1 128.543} C_DIS
LIN {X 0.066,Y -684.631,Z 1161.507,A 0.000,B 0.000,C 90.000,E1 127.317} C_DIS
LIN {X 0.136,Y -688.219,Z 1161.500,A 0.000,B 0.000,C 90.000,E1 125.884} C_DIS
LIN {X -0.130,Y -691.674,Z 1161.492,A 0.000,B 0.000,C 90.000,E1 124.485} C_DIS
LIN {X 0.012,Y -694.457,Z 1161.485,A 0.000,B 0.000,C 90.000,E1 123.293} C_DIS
LIN {X 0.156,Y -696.574,Z 1161.480,A 0.000,B 0.000,C 90.000,E1 122.339} C_DIS
LIN {X -0.290,Y -698.046,Z 1161.476,A 0.000,B 0.000,C 90.000,E1 121.671} C_DIS
LIN {X 0.156,Y -700.289,Z 1161.469,A 0.000,B 0.000,C 90.000,E1 120.463} C_DIS
LIN {X 0.286,Y -702.336,Z 1161.463,A 0.000,B 0.000,C 90.000,E1 119.283} C_DIS
LIN {X -0.169,Y -704.412,Z 1161.456,A 0.000,B 0.000,C 90.000,E1 118.153} C_DIS
